Yaskawa INFORM job: OK_R2_O29-32(90,0_180)OKKR_HARDO.JBI

/JOB
//NAME OK_R2_O29-32(90,0_180)OKKR_HARDO
///FOLDERNAME X4
//POS
///NPOS 481,481,481,29,0,0
///TOOL 0
///POSTYPE PULSE
///PULSE
C00000=-97132,-107765,-123812,202,48316,-59447
C00001=-96375,-92560,-98278,-24892,54395,-33522
C00002=-118989,-99090,-96496,-10423,45001,-41425
C00003=-119482,-98696,-96132,-10013,44918,-41650
C00004=-120044,-95875,-95039,-9417,45618,-41989
C00005=-120040,-96488,-95280,-9446,45452,-41970
C00006=-120040,-96349,-93513,-9613,44449,-41863
C00007=-116902,-102455,-99217,-12157,45235,-40465
C00008=-92713,-84433,-91012,-29057,58273,-28062
C00009=-92713,-84514,-90161,-29225,57775,-27916
C00010=-92713,-84433,-91012,-29057,58273,-28062
C00011=-94031,-81016,-89513,-28080,58570,-28717
C00012=-92713,-84433,-91012,-29057,58273,-28062
C00013=-90703,-81163,-89579,-29929,59661,-27598
C00014=-92713,-84433,-91012,-29057,58273,-28062
C00015=-92432,-93178,-97379,-29384,57863,-27818
C00016=-124148,-115404,-96380,35354,30522,-76988
C00017=-124343,-116589,-99678,31918,27003,-75506
C00018=-121380,-108057,-94385,26950,26949,-73057
C00019=-119584,-104006,-91933,24006,26917,-71617
C00020=-119584,-103646,-90714,24467,26399,-71847
C00021=-119584,-104006,-91933,24006,26917,-71617
C00022=-119620,-100131,-90508,23194,27949,-71207
C00023=-120534,-102543,-91401,24964,27586,-72076
C00024=-122455,-107025,-93629,28318,27362,-73726
C00025=-122455,-106023,-90592,29616,26170,-74375
C00026=-120621,-104452,-90033,26656,25963,-72920
C00027=-122455,-106023,-90592,29616,26170,-74375
C00028=-124343,-116589,-99678,31918,27003,-75506
C00029=-121196,-113012,-111121,15968,43333,-61367
C00030=-113176,-99870,-108783,-18970,68338,-28733
C00031=-120594,-112521,-105960,-11204,51151,-28139
C00032=-122756,-104132,-102044,-9486,52748,-29227
C00033=-121295,-102030,-101271,-10379,53522,-28693
C00034=-122756,-104132,-102044,-9486,52748,-29227
C00035=-120055,-113496,-105331,-11710,50355,-27811
C00036=-117525,-106832,-103510,-13014,52989,-27048
C00037=-118169,-104316,-102602,-12476,53606,-27398
C00038=-117525,-106832,-103510,-13014,52989,-27048
C00039=-120055,-113496,-105331,-11710,50355,-27811
C00040=-122277,-105580,-101993,-9905,52039,-28956
C00041=-122277,-105483,-101030,-9979,51504,-28904
C00042=-122277,-105580,-101993,-9905,52039,-28956
C00043=-114234,-96976,-102629,-20681,62688,-27649
C00044=-111778,-96221,-107052,-21188,70616,-22267
C00045=-117350,-114999,-95956,-52919,38370,-55080
C00046=-108972,-69269,-80208,-51978,72625,-32902
C00047=-109543,-61925,-78651,-49562,78172,-29234
C00048=-109543,-62109,-77971,-49635,77832,-29052
C00049=-109543,-61925,-78651,-49562,78172,-29234
C00050=-110239,-61041,-78189,-49323,77924,-29446
C00051=-109543,-61925,-78651,-49562,78172,-29234
C00052=-107063,-66961,-84785,-50173,80254,-29118
C00053=-90901,-32599,-64406,-54667,92064,-27755
C00054=-92412,-28582,-59178,-54201,90556,-27610
C00055=-92412,-29145,-58034,-54170,89959,-27242
C00056=-92412,-28659,-59030,-54195,90478,-27561
C00057=-93599,-27197,-58027,-53876,89920,-27837
C00058=-92412,-28659,-59030,-54195,90478,-27561
C00059=-94015,-33926,-70364,-53928,92204,-29442
C00060=-96981,-29734,-65408,-52966,90116,-29668
C00061=-96981,-30385,-64512,-52944,89568,-29346
C00062=-96981,-29921,-65159,-52958,89962,-29578
C00063=-97341,-27509,-63519,-52853,89918,-29730
C00064=-96981,-29921,-65159,-52958,89962,-29578
C00065=-83985,-34763,-79826,-57770,100542,-29760
C00066=-119227,-121429,-124211,-4290,80037,5069
C00067=-103198,-96938,-112022,-8857,86341,9990
C00068=-104928,-94630,-110553,-8370,86444,9424
C00069=-105210,-91425,-109287,-8287,87275,9277
C00070=-105152,-92089,-109552,-8304,87105,9308
C00071=-105152,-92773,-108542,-8308,86142,9373
C00072=-104752,-96369,-111669,-8420,86257,9494
C00073=-93824,-83108,-104490,4346,83202,15848
C00074=-94227,-80625,-103370,4481,83809,15742
C00075=-95161,-74712,-100714,4798,85256,15503
C00076=-95037,-75505,-101078,4756,85066,15534
C00077=-95037,-76584,-99812,4762,83737,15482
C00078=-95852,-86288,-106522,5052,82929,15193
C00079=-119227,-121429,-124211,-4290,80037,5069
C00080=-108780,-117808,-111617,-31391,23506,27123
C00081=-87227,-129275,-103249,-15171,52693,43306
C00082=-62701,-112417,-81564,-27325,55133,54084
C00083=-102122,-48912,-69312,-5951,70900,35879
C00084=-115730,-7694,-35577,433,70873,-75154
C00085=-117065,58625,15220,1046,73703,-75581
C00086=-145520,63530,20841,13896,75272,-84857
C00087=-144593,33918,-9965,-2110,74261,-87786
C00088=-145469,31320,-10101,-1692,72990,-88049
C00089=-145469,30699,-8934,-1700,71953,-88037
C00090=-145469,30866,-9263,-1698,72241,-88041
C00091=-145880,26405,-13670,-1493,72653,-88180
C00092=-145880,26179,-13238,-1495,72270,-88176
C00093=-145579,28506,-10956,-1645,72067,-88074
C00094=-145661,28530,-12807,-1597,73217,-88116
C00095=-144591,77564,35073,-17956,86562,-90701
C00096=-144815,78144,37521,-17912,85364,-90602
C00097=-144815,77832,38454,-17925,84664,-90498
C00098=-144815,77924,38162,-17920,84880,-90530
C00099=-143930,80933,41834,-18166,84388,-90155
C00100=-143930,80814,42260,-18173,84080,-90109
C00101=-144274,79788,41005,-18076,84241,-90251
C00102=-144021,80584,40299,-18125,85099,-90292
C00103=-142778,71394,29201,-18425,87369,-90210
C00104=-142778,70963,30227,-18429,86558,-90088
C00105=-142778,71046,30015,-18428,86723,-90113
C00106=-141980,74470,34104,-18641,86176,-89759
C00107=-141980,74364,34402,-18643,85951,-89725
C00108=-142286,73285,33109,-18561,86114,-89854
C00109=-142258,74173,32193,-18559,87090,-89993
C00110=-151142,95382,53861,9912,94501,-89436
C00111=-151142,95214,54369,9904,94108,-89467
C00112=-151142,94960,55250,9895,93443,-89520
C00113=-151142,95064,54871,9900,93726,-89497
C00114=-151832,99566,60657,9969,92580,-89818
C00115=-151832,99473,61122,9966,92251,-89844
C00116=-151679,98392,59730,9950,92531,-89770
C00117=-151679,98651,58626,9962,93331,-89705
C00118=-139326,110012,65153,-7943,96581,-88072
C00119=-139426,116179,73372,-7897,94700,-87984
C00120=-139426,115886,74309,-7888,93978,-87938
C00121=-139426,116062,73720,-7895,94427,-87966
C00122=-140236,121957,81659,-7780,92511,-88115
C00123=-140236,121844,82405,-7775,91998,-88082
C00124=-140074,120418,80479,-7799,92463,-88057
C00125=-140074,120860,78539,-7816,93872,-88145
C00126=-141384,30046,-16215,-3642,76218,-86818
C00127=-144769,2915,-41310,-1997,77613,-87897
C00128=-120497,-21208,-21286,5945,66983,1716
C00129=-120331,-15331,-14033,5953,65534,1703
C00130=-120268,-12560,-10010,5981,64483,1671
C00131=-120268,-12013,-7946,6027,63500,1622
C00132=-120268,-12272,-8910,6006,63957,1643
C00133=-120268,-12272,-8910,6006,63957,1643
C00134=-120271,-10596,-7611,6006,64020,1643
C00135=-120265,-13710,-11092,5976,64558,1676
C00136=-121090,-15095,-12910,6234,65025,1394
C00137=-122392,-36893,-37139,6496,68816,1124
C00138=-103008,-20958,-23789,-34380,46191,-50944
C00139=-106920,-17705,-17148,-23301,36916,-65920
C00140=-100038,-3407,1736,-8309,24573,-69609
C00141=-100051,-3014,2749,-8424,24152,-69554
C00142=-100051,-2528,4297,-8659,23456,-69437
C00143=-99986,-3534,2326,-8528,24154,-69501
C00144=-100190,-1879,3683,-8197,24147,-69667
C00145=-100051,-3014,2749,-8424,24152,-69554
C00146=-107520,-15673,-12264,3373,26664,-75475
C00147=-107604,-14630,-9438,-26327,31803,-64502
C00148=-107301,-12783,-11511,-23446,35942,-65836
C00149=-106944,-14381,-11463,-24264,35264,-65385
C00150=-107257,-12837,-10189,-14623,32274,-69602
C00151=-111525,-14589,-10078,-816,28523,-72551
C00152=-98801,-12889,-18000,4905,35451,-65199
C00153=-115508,-28515,-28430,43638,36769,-74115
C00154=-104252,-46667,-49928,-23147,42547,-66097
C00155=-139326,111643,62701,-7999,98906,-88222
C00156=-140217,96503,46831,-7956,100791,-62986
C00157=-145074,69745,16622,-2645,91472,-63331
C00158=-144953,70943,20162,-2680,89915,-63261
C00159=-144922,69779,18776,-2690,90171,-63257
C00160=-144922,69779,18776,-2690,90171,-63257
C00161=-145083,66914,15382,-2644,90782,-63319
C00162=-137468,95477,49594,-19726,99949,-65005
C00163=-137749,101548,57639,-20808,101771,-65556
C00164=-141788,85517,37198,-20977,104871,-67541
C00165=-141788,85517,37198,-20977,104871,-67541
C00166=-141697,80573,32373,-24906,103800,-68015
C00167=-141133,64860,16683,-29804,96213,-66902
C00168=-143290,70938,23843,-29251,94388,-67208
C00169=-143290,72189,22259,-29351,95808,-67570
C00170=-136972,39162,-14968,-31401,103005,-67268
C00171=-136972,39162,-14968,-31401,103005,-67268
C00172=-104252,-46667,-49928,-23147,42547,-66097
C00173=-79661,-64382,-64322,-40022,51624,-56449
C00174=-25614,-129739,-89176,-60277,72547,-35569
C00175=-79661,-64382,-64322,-40022,51624,-56449
C00176=-120757,-91510,-125291,13460,57469,62186
C00177=-120699,-18778,-86977,11996,70937,63715
C00178=-120626,-71428,-80514,17274,40782,59546
C00179=-119608,-71223,-77796,25261,41295,55541
C00180=-118939,-66183,-73787,24596,41210,55877
C00181=-120629,-71631,-77769,17920,39069,59168
C00182=-120359,-74344,-77822,18174,37713,59000
C00183=-130492,-64065,-72622,39267,48666,48449
C00184=-128767,-64530,-72039,39655,46741,50471
C00185=-122213,-56683,-67868,39757,48514,50554
C00186=-119025,-61972,-83652,25821,56823,82211
C00187=-119200,-79046,-90724,17013,50162,51422
C00188=-120627,-71422,-82568,-22551,39281,-72893
C00189=-120626,-71781,-79821,-23470,37548,-72366
C00190=-120451,-70478,-78279,-23795,37340,-72196
C00191=-120359,-74605,-80000,-24468,36394,-71829
C00192=-120633,-71786,-79901,-23439,37590,-72383
C00193=-120966,-71169,-78914,-23220,37205,-72458
C00194=-120627,-71746,-82478,-22655,39075,-72833
C00195=-120628,-68509,-91693,-24468,73270,-29259
C00196=-120628,-69110,-90711,-24576,72437,-29080
C00197=-120650,-67557,-87939,-24676,71616,-28918
C00198=-120635,-69084,-90779,-24566,72485,-29092
C00199=-120360,-72648,-91234,-24892,71146,-28701
C00200=-102891,-55002,-81397,-31881,79379,-24336
C00201=-98614,-51013,-79162,-33441,81477,-23356
C00202=-110216,-66091,-87232,-17856,68486,-33346
C00203=-120628,-67132,-93536,-6272,76376,-26037
C00204=-120629,-65307,-95540,-6224,78533,-26146
C00205=-125976,-49581,-89047,24033,107700,-27220
C00206=-114932,-69047,-98963,12803,96211,-16970
C00207=-121913,-67019,-96424,19539,98441,-21657
C00208=-120636,-64508,-96476,19357,99419,-21079
C00209=-115636,-66806,-97970,12989,96839,-17125
C00210=-122763,-41192,-84008,14889,102356,-18715
C00211=-119690,-45533,-86635,11059,99611,-14244
C00212=-123247,-59553,-98781,12453,98224,-12183
C00213=-120629,-65231,-95763,5470,82909,-26902
C00214=-114225,-78059,-113057,2895,86652,-24852
C00215=-100902,-64627,-95050,-11985,78171,-15678
C00216=-98861,-75542,-94548,-15732,66869,-13224
C00217=-119874,-71154,-93232,19306,73218,3187
C00218=-121912,-70007,-92672,20214,73908,2597
C00219=-98680,-77069,-90223,-16254,63590,-12696
C00220=-96345,-50788,-86680,-18048,88539,-14542
C00221=-93223,-76561,-100164,-23339,71866,-11449
C00222=-120630,-61713,-98239,-7195,94993,11495
C00223=-120629,-64150,-96408,-7165,92633,11631
C00224=-127375,-45154,-88676,-4909,106126,9193
C00225=-120636,-64104,-96466,-7164,92690,11625
C00226=-119876,-67808,-97008,-7371,91195,11945
C00227=-122268,-40179,-85765,-5907,107177,10698
C00228=-117984,-41448,-85856,-6781,104340,12121
C00229=-117785,-40415,-85699,-6838,104785,12155
C00230=-118921,-47757,-88901,-6950,100752,11907
C00231=-128083,-66216,-96645,-288,90786,4689
C00232=-127344,-66265,-96731,-512,90816,4915
C00233=-120629,-63706,-96407,-7167,92858,11618
C00234=-119771,-61779,-98541,-7450,95212,11740
C00235=-113204,-65987,-111954,-20711,103856,-62714
C00236=-120630,-56479,-101004,-18441,100644,-64439
C00237=-137856,-73372,-107086,809,89532,-64747
C00238=-119374,-56629,-99297,-18722,99813,-63925
C00239=-120637,-56952,-100808,-18413,100297,-64387
C00240=-141222,-46996,-93568,2005,94815,-65665
C00241=-144586,-98422,-105395,6853,55489,-67509
C00242=-126129,-101623,-112002,-18280,57665,-60270
C00243=-107171,-88917,-111068,-40561,70673,-56675
C00244=-99343,-43314,-99502,-42439,86261,-59904
C00245=-52791,5163,-64646,-46831,92051,-59410
C00246=3643,-76224,-106676,19950,71810,76872
C00247=-31759,-97415,-96886,-14116,45711,48381
C00248=-44548,-99394,-97233,-12419,44266,52870
C00249=-91182,-106612,-98498,-6229,38996,69241
C00250=-120252,-111112,-99286,-2370,35711,79446
C00251=-120252,-111112,-99286,-2370,35711,79446
C00252=-122061,-111349,-89048,-12693,25666,-59648
C00253=-121671,-62095,-66353,-9610,36862,-61269
C00254=-121347,-21258,-21397,-11816,30334,-60091
C00255=-120891,-15529,-14207,-12963,28955,-59505
C00256=-120717,-13203,-11253,-13455,28377,-59255
C00257=-120568,-11431,-9889,-13625,28472,-59171
C00258=-120717,-13203,-11253,-13455,28377,-59255
C00259=-120696,-12930,-10087,-13737,27819,-59112
C00260=-120692,-12567,-8711,-14046,27176,-58956
C00261=-120696,-12930,-10087,-13737,27819,-59112
C00262=-120870,-15275,-13061,-13229,28399,-59370
C00263=-123043,5425,8644,-60342,36239,-52197
C00264=-124447,11447,16156,-60569,34992,-52124
C00265=-124447,11983,17788,-61490,34623,-51621
C00266=-127145,7414,15485,-62450,27197,-51222
C00267=-127103,8624,16548,-62533,27208,-51178
C00268=-127127,7743,15901,-62612,27166,-51140
C00269=-124895,-3553,-1899,-45295,28876,-55547
C00270=-121324,-21046,-20294,-12047,29779,-59971
C00271=-121671,-62095,-66353,-9610,36862,-61269
C00272=-122061,-111349,-89048,-12693,25666,-59648
C00273=-120249,-110580,-95500,-2498,33656,79516
C00274=-120367,-55464,-65807,-1899,43695,79179
C00275=-120372,-19909,-20534,-2331,34109,79427
C00276=-120603,-14858,-13386,-2171,32301,79344
C00277=-118432,-12836,-10242,-4853,31501,80756
C00278=-118432,-12391,-8558,-4969,30699,80814
C00279=-118432,-12586,-9286,-4918,31044,80789
C00280=-118432,-12586,-9286,-4918,31044,80789
C00281=-118451,-11211,-8225,-4888,31096,80773
C00282=-120719,-12556,-10288,-2076,31575,79294
C00283=-120630,-14625,-13229,-2138,32324,79327
C00284=-131566,-7566,-2012,56880,47864,36778
C00285=-127270,2858,10417,64219,55978,24180
C00286=-127270,2872,10457,64230,55970,24171
C00287=-127270,3275,11649,64548,55732,23910
C00288=-127279,2816,10434,64241,55969,24162
C00289=-127226,4202,11617,64241,55929,24162
C00290=-127288,2760,10411,64252,55968,24153
C00291=-139196,1750,6280,64814,64625,23032
C00292=-119950,-29718,-27457,-2865,33344,79709
C00293=-120367,-55464,-65807,-1899,43695,79179
C00294=-120071,-144849,-99630,-4685,18622,80601
C00295=-120101,-156003,-112174,-4198,20603,80368
C00296=-118703,-129435,-118376,-15737,33464,74082
C00297=-118229,-124990,-122609,-18843,37087,72450
C00298=-117709,-116078,-100914,-29615,27785,74634
C00299=-121884,-95901,-99968,19866,48605,45126
C00300=-120671,-70136,-84949,27990,60023,38564
C00301=-120478,-67274,-83298,27761,60367,38737
C00302=-120671,-68730,-84259,27912,60289,38637
C00303=-120481,-64965,-83246,27119,62754,39366
C00304=-120481,-65408,-81931,27360,61828,39126
C00305=-121686,-66768,-84557,27809,63026,38954
C00306=-141024,-58078,-80968,36822,71957,33892
C00307=-140832,-52974,-76512,36762,71783,33908
C00308=-140832,-53417,-75497,36922,71094,33665
C00309=-140832,-52974,-76512,36762,71783,33908
C00310=-140279,-50808,-75283,36453,71852,34159
C00311=-140832,-52974,-76512,36762,71783,33908
C00312=-109942,-69794,-83321,-14013,53448,56252
C00313=-112063,-69620,-83237,-12481,53147,55418
C00314=-109971,-72059,-85461,-13968,53588,56219
C00315=-110807,-74146,-92563,-12442,56365,55924
C00316=-138671,-88440,-95611,17208,48170,52520
C00317=-138671,-88615,-94297,17448,47310,52358
C00318=-138671,-88440,-95611,17208,48170,52520
C00319=-138502,-86929,-95389,16910,48750,52704
C00320=-138041,-84511,-94358,16397,49242,52997
C00321=-138502,-86929,-95389,16910,48750,52704
C00322=-119374,-94871,-99184,-14699,45596,69062
C00323=-119374,-95024,-95430,-15324,43285,69457
C00324=-120961,-93958,-95008,-13845,43283,68674
C00325=-119374,-95024,-95430,-15324,43285,69457
C00326=-119544,-103546,-104622,-14834,44490,69166
C00327=-118175,-83390,-115370,-9254,78664,2265
C00328=-136131,-54129,-95643,4560,92395,119
C00329=-136131,-54129,-95643,4560,92395,119
C00330=-136131,-54129,-95643,4560,92395,119
C00331=-136131,-55910,-94548,4553,90811,61
C00332=-136131,-54129,-95643,4560,92395,119
C00333=-118826,-50989,-93921,-11407,94620,13199
C00334=-119876,-53326,-92440,-11017,92423,13086
C00335=-120690,-52300,-91874,-10745,92506,12834
C00336=-119876,-53326,-92440,-11017,92423,13086
C00337=-118826,-50270,-94307,-11422,95216,13144
C00338=-141793,-55820,-97332,7512,93105,-2300
C00339=-140356,-59957,-95696,6990,89886,-2061
C00340=-139743,-58912,-95151,6779,90039,-1868
C00341=-140356,-59957,-95696,6990,89886,-2061
C00342=-140356,-55082,-98612,7026,94155,-1823
C00343=-131844,-82412,-106901,19181,77049,14413
C00344=-121763,-121440,-108343,34263,48676,32319
C00345=-121436,-111193,-102207,33362,49794,32929
C00346=-120328,-103716,-97102,32376,49958,33559
C00347=-120328,-103424,-95545,32743,49272,33305
C00348=-120328,-103597,-96437,32532,49662,33450
C00349=-119706,-101713,-95741,31911,49887,33849
C00350=-120328,-103597,-96437,32532,49662,33450
C00351=-120421,-109652,-101209,32668,49551,33360
C00352=-120678,-119715,-107328,33483,48463,32809
C00353=-145717,-65257,-81010,41655,68644,28827
C00354=-145541,-64355,-79967,41625,68428,28817
C00355=-145541,-64661,-78699,41864,67717,28513
C00356=-145541,-64450,-79596,41693,68217,28727
C00357=-144419,-63348,-79027,41165,67869,29094
C00358=-145541,-64450,-79596,41693,68217,28727
C00359=-144489,-68274,-88356,40433,70363,30088
C00360=-140701,-65348,-85833,38739,68695,31071
C00361=-140701,-65803,-84785,38949,68003,30804
C00362=-140701,-65400,-85721,38761,68620,31042
C00363=-140042,-62987,-84490,38345,68721,31364
C00364=-140701,-65400,-85721,38761,68620,31042
C00365=-129105,-89797,-100104,-8257,42122,-63791
C00366=-127638,-62786,-75319,-9961,40926,-62941
C00367=-127541,-60842,-73212,-10119,40642,-62858
C00368=-127452,-58887,-72168,-10136,41010,-62858
C00369=-127541,-60842,-73212,-10119,40642,-62858
C00370=-127484,-59721,-71596,-10263,40237,-62779
C00371=-127484,-59825,-70645,-10399,39608,-62699
C00372=-127484,-59721,-71596,-10263,40237,-62779
C00373=-128516,-69367,-82634,-8882,41931,-63486
C00374=-136804,-49406,-65089,-22327,37576,-67328
C00375=-138093,-44400,-58341,-21720,35770,-67534
C00376=-137893,-42671,-57282,-21821,36047,-67500
C00377=-138034,-43342,-57719,-21701,35939,-67550
C00378=-137984,-43593,-56312,-22278,35025,-67233
C00379=-137984,-43463,-57769,-21774,35919,-67515
C00380=-121497,-78215,-85327,-19946,40083,-59616
C00381=-120626,-71657,-80701,-17243,40860,-59361
C00382=-126255,-72821,-79643,-11943,38658,-61920
C00383=-124460,-69554,-75696,-14032,38208,-60874
C00384=-120888,-74575,-78008,-18145,37790,-58814
C00385=-120633,-71857,-77956,-17876,39147,-58988
C00386=-120627,-71204,-76479,-18098,38609,-58863
C00387=-136164,-60832,-69738,-17624,37003,-72099
C00388=-124488,-74552,-79755,-29777,39497,-66170
C00389=-118213,-106277,-106559,-35084,42029,-63565
C00390=-120627,-70570,-83191,7863,37643,76584
C00391=-120626,-71021,-80486,8216,35764,76386
C00392=-117835,-70487,-78994,2708,35489,78081
C00393=-120887,-73898,-80698,8807,34458,76086
C00394=-120633,-71014,-80560,8214,35814,76388
C00395=-120357,-69871,-78574,5676,35674,76676
C00396=-149434,-47635,-66681,32878,46415,64025
C00397=-156080,-38551,-61157,37208,50074,62118
C00398=-120626,-71358,-80242,8280,35444,76351
C00399=-120627,-70947,-82965,7922,37313,76550
C00400=-120635,-68263,-89533,19357,55237,54189
C00401=-120627,-69277,-87249,27960,61590,38909
C00402=-120627,-70131,-84728,28472,59826,38424
C00403=-119745,-63249,-82789,26446,65626,40301
C00404=-120887,-73269,-85067,29013,58674,37985
C00405=-120633,-70114,-84797,28462,59873,38435
C00406=-120443,-58955,-81680,26193,68992,40844
C00407=-137016,-48093,-75675,33483,76149,36536
C00408=-111378,-73522,-86374,8880,55488,45224
C00409=-108292,-90151,-101040,6716,55677,46453
C00410=-104551,-107393,-114036,4170,54574,47870
C00411=-131132,-52506,-88181,-2999,76585,58563
C00412=-128416,-45796,-82269,-5250,83117,42213
C00413=-120634,-69367,-86746,-19850,61513,61572
C00414=-119352,-71200,-86390,-20819,60725,62219
C00415=-124049,-46051,-81029,-10377,81461,42067
C00416=-121481,-32611,-71357,-8547,80518,38471
C00417=-129432,-34048,-72513,3927,79787,30181
C00418=-133185,-27484,-76607,10911,90885,32661
C00419=-131562,-31841,-87200,10336,94922,33460
C00420=-120628,-67882,-90305,8002,60955,27137
C00421=-120628,-68780,-88641,8118,59484,27029
C00422=-119184,-68852,-87338,7230,58521,27500
C00423=-119351,-70586,-88688,7347,58476,27433
C00424=-121372,-71710,-89222,8706,58421,26669
C00425=-119224,-70326,-83140,7530,55210,27256
C00426=-118796,-48871,-84615,7155,80182,30422
C00427=-125592,-51833,-97720,10091,87276,28906
C00428=-113783,-56439,-81210,15698,57996,69309
C00429=-107790,-54952,-79381,11557,56703,71425
C00430=-114138,-25426,-67877,22136,88341,34287
C00431=-121370,-73680,-74765,39382,39185,61177
C00432=-120632,-71435,-74935,37828,39854,62032
C00433=-120118,-28476,-67262,26234,84322,31994
C00434=-128183,-20881,-60116,35034,87592,29156
C00435=-128620,-20492,-59969,35459,87655,29119
C00436=-131561,-17349,-57221,36148,87598,28432
C00437=-145073,1746,-39674,39691,86205,25187
C00438=-146718,4880,-36652,40179,85809,24767
C00439=-152046,17466,-29664,47680,97969,20185
C00440=-155175,14277,-38805,49221,102130,20939
C00441=-135677,-24502,-83351,29476,105612,50888
C00442=-120631,-49325,-102634,14154,102303,71085
C00443=-120630,-54638,-100904,13945,98616,70657
C00444=-113110,-76964,-106909,6133,84021,70452
C00445=-120637,-55119,-100712,13931,98263,70614
C00446=-121882,-54885,-99226,14292,97671,70180
C00447=-108261,-50195,-93515,4199,89241,72102
C00448=-118173,-67191,-91447,22538,66327,68916
C00449=-120627,-69075,-88308,30031,58405,66774
C00450=-120628,-67609,-91029,29341,60528,67400
C00451=-120651,-137986,-128118,34242,49089,63541
C00452=-120704,-83666,-109294,28636,63184,68115
C00453=-120704,-83666,-109294,28636,63184,68115
C00454=-122061,-111349,-89048,-12693,25666,-59648
C00455=-121671,-62095,-66353,-9610,36862,-61269
C00456=-120675,-12683,-10165,-1101,31339,-85533
C00457=-117312,-15222,-7734,-15098,24829,-82061
C00458=-120855,-14769,-11753,-884,31242,-85646
C00459=-120680,-13066,-11724,-1072,32101,-85548
C00460=-110921,-9380,-5536,-39323,36544,-54600
C00461=-105611,16644,27067,-74678,55970,-29641
C00462=-105060,15092,17806,-65581,60394,-35506
C00463=-113952,17541,-9445,-35713,50265,-81352
C00464=-121726,-68659,-62259,-14447,23269,-58731
C00465=-122061,-111349,-89048,-12693,25666,-59648
C00466=-120249,-110580,-95500,-2498,33656,79516
C00467=-120367,-55464,-65807,-1899,43695,79179
C00468=-123079,18123,-5334,37346,69821,35077
C00469=-120790,5622,-11235,35661,58510,35599
C00470=-123082,18120,-5282,37355,69796,35066
C00471=-123254,15918,-6072,37557,69350,34829
C00472=-101635,-726,-13913,25769,46964,40903
C00473=-122250,26655,19444,63036,59530,30813
C00474=-129965,36435,30593,70202,68747,28349
C00475=-135677,36825,21549,57633,74723,28944
C00476=-134949,-3767,-37487,36447,81076,35091
C00477=-139267,-30752,-53917,52477,61088,25483
C00478=-156581,-111669,-93710,65875,62680,14502
C00479=-153491,-118067,-95704,59271,58057,20364
C00480=-32064,-128753,-95704,15399,77815,-718
BC00000=40633,757095,1075175
BC00001=40600,786248,1075175
BC00002=40600,786248,1075175
BC00003=40600,786248,1075175
BC00004=40600,786248,1075175
BC00005=40600,786248,1075175
BC00006=40600,786248,1075175
BC00007=40600,786248,1075175
BC00008=40594,791778,1075175
BC00009=40594,791778,1075175
BC00010=40594,791778,1075175
BC00011=40594,791778,1075175
BC00012=40594,791778,1075175
BC00013=40594,791778,1075175
BC00014=40594,791778,1075175
BC00015=40594,791778,1075175
BC00016=40594,791778,1075175
BC00017=50995,786704,1075175
BC00018=50995,786704,1075175
BC00019=50995,786704,1075175
BC00020=50995,786704,1075175
BC00021=50995,786704,1075175
BC00022=50995,786704,1075175
BC00023=50995,786704,1075175
BC00024=50995,786704,1075175
BC00025=50995,786704,1075175
BC00026=50995,786704,1075175
BC00027=50995,786704,1075175
BC00028=50995,786704,1075175
BC00029=64165,785759,1075175
BC00030=97726,783351,1075175
BC00031=97726,783351,1075175
BC00032=97726,783351,1075175
BC00033=97726,783351,1075175
BC00034=97726,783351,1075175
BC00035=97726,783351,1075175
BC00036=97726,783351,1075175
BC00037=97726,783351,1075175
BC00038=97726,783351,1075175
BC00039=97726,783351,1075175
BC00040=97726,783351,1075175
BC00041=97726,783351,1075175
BC00042=97726,783351,1075175
BC00043=97726,783351,1075175
BC00044=97726,783351,1075175
BC00045=161258,787851,1075175
BC00046=161258,787851,1075175
BC00047=161258,787851,1075175
BC00048=161258,787851,1075175
BC00049=161258,787851,1075175
BC00050=161258,787851,1075175
BC00051=161258,787851,1075175
BC00052=161258,787851,1075175
BC00053=161258,787851,1075175
BC00054=161258,787851,1075175
BC00055=161258,787851,1075175
BC00056=161258,787851,1075175
BC00057=161258,787851,1075175
BC00058=161258,787851,1075175
BC00059=161258,787851,1075175
BC00060=161258,787851,1075175
BC00061=161258,787851,1075175
BC00062=161258,787851,1075175
BC00063=161258,787851,1075175
BC00064=161258,787851,1075175
BC00065=161258,787851,1075175
BC00066=272656,866721,1075175
BC00067=272656,866721,1075175
BC00068=272656,866721,1075175
BC00069=272656,866721,1075175
BC00070=272656,866721,1075175
BC00071=272656,866721,1075175
BC00072=272656,866721,1075175
BC00073=272656,866721,1075175
BC00074=272656,866721,1075175
BC00075=272656,866721,1075175
BC00076=272656,866721,1075175
BC00077=272656,866721,1075175
BC00078=272656,866721,1075175
BC00079=272656,866721,1075175
BC00080=276508,696729,1075050
BC00081=283938,685942,1074810
BC00082=283938,717840,610142
BC00083=283938,747609,176485
BC00084=283938,747609,176485
BC00085=283938,747609,53405
BC00086=343059,747609,53405
BC00087=343059,747609,53405
BC00088=343059,747609,53405
BC00089=343059,747609,53405
BC00090=343059,747609,53405
BC00091=343059,747609,53405
BC00092=343059,747609,53405
BC00093=343059,747609,53405
BC00094=343059,747609,53405
BC00095=343059,747609,53405
BC00096=343059,747609,53405
BC00097=343059,747609,53405
BC00098=343059,747609,53405
BC00099=343059,747609,53405
BC00100=343059,747609,53405
BC00101=343059,747609,53405
BC00102=343059,747609,53405
BC00103=343059,747609,53405
BC00104=343059,747609,53405
BC00105=343059,747609,53405
BC00106=343059,747609,53405
BC00107=343059,747609,53405
BC00108=343059,747609,53405
BC00109=343059,747609,53405
BC00110=343059,747609,53405
BC00111=343059,747609,53405
BC00112=343059,747609,53405
BC00113=343059,747609,53405
BC00114=343059,747609,53405
BC00115=343059,747609,53405
BC00116=343059,747609,53405
BC00117=343059,747609,53405
BC00118=343059,747609,24
BC00119=343059,747609,24
BC00120=343059,747609,24
BC00121=343059,747609,24
BC00122=343059,747609,24
BC00123=343059,747609,24
BC00124=343059,747609,24
BC00125=343059,747609,24
BC00126=343059,747609,53405
BC00127=343059,747609,53405
BC00128=272784,788172,221315
BC00129=272784,788172,221315
BC00130=272784,788172,221315
BC00131=272784,788172,221315
BC00132=272784,788172,221315
BC00133=272784,788172,221315
BC00134=272784,788172,221315
BC00135=272784,788172,221315
BC00136=272784,788172,221315
BC00137=272784,788172,221315
BC00138=262280,759997,129875
BC00139=260494,755206,114324
BC00140=260786,755989,116866
BC00141=260786,755989,116866
BC00142=260786,755989,116866
BC00143=260786,755989,116866
BC00144=260786,755989,116866
BC00145=260786,755989,116866
BC00146=260786,755989,116866
BC00147=260462,756705,106964
BC00148=260456,756989,105568
BC00149=260456,756989,105568
BC00150=253777,756505,101682
BC00151=288441,762581,102049
BC00152=263875,774786,46208
BC00153=263467,774501,47249
BC00154=260494,755206,114324
BC00155=343059,747609,24
BC00156=344552,769122,24
BC00157=344552,769122,24
BC00158=344552,769122,24
BC00159=344552,769122,24
BC00160=344552,769122,24
BC00161=344552,769122,24
BC00162=344552,769122,24
BC00163=344552,769122,24
BC00164=344552,769122,24
BC00165=344552,769122,24
BC00166=344552,769122,24
BC00167=344552,769122,24
BC00168=344552,769122,24
BC00169=344552,769122,24
BC00170=344552,769122,24
BC00171=344552,769122,24
BC00172=260494,755206,114324
BC00173=260494,678873,114324
BC00174=260494,678873,389237
BC00175=260494,678873,1074810
BC00176=249358,694721,1075175
BC00177=249358,736986,1075175
BC00178=249358,791546,1075175
BC00179=248933,799175,1075175
BC00180=248933,799175,1075175
BC00181=248933,799175,1075175
BC00182=248933,799175,1075175
BC00183=303936,808747,1075173
BC00184=301664,808908,1075173
BC00185=301664,808908,1075173
BC00186=278558,810544,1075175
BC00187=259247,802769,1075175
BC00188=179692,770739,1075175
BC00189=178037,775961,1075175
BC00190=177375,778050,1075175
BC00191=177375,778050,1075175
BC00192=177375,778050,1075175
BC00193=105009,765455,1075171
BC00194=106185,757956,1075175
BC00195=70430,778998,1075175
BC00196=70141,784459,1075175
BC00197=70031,786589,1075172
BC00198=70026,786643,1075175
BC00199=70026,786643,1075175
BC00200=71134,786838,1075175
BC00201=71134,786838,1075175
BC00202=71134,786838,1075175
BC00203=80371,790898,1075175
BC00204=79285,785365,1075175
BC00205=47064,807646,1075175
BC00206=47064,807646,1075175
BC00207=47306,807824,1075175
BC00208=47306,807824,1075175
BC00209=47064,807646,1075175
BC00210=47064,807646,1075175
BC00211=47064,807646,1075175
BC00212=47064,807646,1075175
BC00213=54175,793583,1075175
BC00214=54175,793583,1075175
BC00215=54992,769398,1075175
BC00216=54992,769398,1075175
BC00217=54992,769398,1075175
BC00218=54992,769398,1075175
BC00219=54992,769398,1075175
BC00220=54992,769398,1075175
BC00221=54992,769398,1075175
BC00222=110304,782517,1075175
BC00223=108105,787545,1075175
BC00224=107226,789556,1075175
BC00225=107226,789556,1075175
BC00226=107226,789556,1075175
BC00227=107226,789556,1075175
BC00228=107227,789556,1075174
BC00229=107227,789556,1075174
BC00230=127545,800970,1075174
BC00231=170992,825380,1075175
BC00232=170992,825380,1075175
BC00233=172064,823477,1075175
BC00234=174263,818448,1075175
BC00235=118984,806720,1075175
BC00236=118671,807322,1075175
BC00237=118546,807563,1075175
BC00238=118546,807563,1075175
BC00239=118546,807563,1075175
BC00240=118546,807563,1075175
BC00241=118546,807563,1075175
BC00242=125414,796325,1075175
BC00243=133048,783833,1075175
BC00244=133048,783833,1075175
BC00245=133048,671052,1075175
BC00246=199464,674570,1075173
BC00247=264750,673287,320956
BC00248=270450,673384,288313
BC00249=291235,673736,169281
BC00250=304191,673956,95082
BC00251=304191,673956,95082
BC00252=164726,705512,84367
BC00253=164726,728796,84367
BC00254=164726,745774,84367
BC00255=164726,745774,84367
BC00256=164726,745774,84367
BC00257=164726,745774,84367
BC00258=164726,745774,84367
BC00259=164726,745774,84367
BC00260=164726,745774,84367
BC00261=164726,745774,84367
BC00262=164726,745774,84367
BC00263=164726,745774,84367
BC00264=164726,745774,84367
BC00265=164726,745774,84367
BC00266=164726,745774,84367
BC00267=164726,745774,84367
BC00268=164726,745774,84367
BC00269=164726,745774,84367
BC00270=164726,745774,84367
BC00271=164726,728796,84367
BC00272=164726,705512,84367
BC00273=304191,706504,95082
BC00274=304191,706504,95082
BC00275=304191,726145,95082
BC00276=304191,726145,95082
BC00277=304191,726145,95082
BC00278=304191,726145,95082
BC00279=304191,726145,95082
BC00280=304191,726145,95082
BC00281=304191,726145,95082
BC00282=304191,726145,95082
BC00283=304191,726145,95082
BC00284=304191,726145,95082
BC00285=304191,726145,95082
BC00286=304191,726145,95082
BC00287=304191,726145,95082
BC00288=304191,726145,95082
BC00289=304191,726145,95082
BC00290=304191,726145,95082
BC00291=304191,726145,95082
BC00292=304191,726145,95082
BC00293=304191,706504,95082
BC00294=304191,706504,95082
BC00295=304191,706504,1074810
BC00296=355942,722834,1075048
BC00297=369200,753216,1075109
BC00298=383735,786522,1075175
BC00299=370224,778181,1075175
BC00300=364232,774482,1075175
BC00301=364232,774482,1075175
BC00302=364232,774482,1075175
BC00303=364232,774482,1075175
BC00304=364232,774482,1075175
BC00305=364232,774482,1075175
BC00306=364232,774482,1075175
BC00307=364232,774482,1075175
BC00308=364232,774482,1075175
BC00309=364232,774482,1075175
BC00310=364232,774482,1075175
BC00311=364232,774482,1075175
BC00312=364232,774482,1075175
BC00313=364232,774482,1075175
BC00314=364232,774482,1075175
BC00315=365231,775099,1075175
BC00316=383734,786522,1075172
BC00317=383734,786522,1075172
BC00318=383734,786522,1075172
BC00319=383734,786522,1075172
BC00320=383734,786522,1075172
BC00321=383734,786522,1075172
BC00322=383735,786522,1075175
BC00323=383735,786522,1075175
BC00324=383735,786522,1075175
BC00325=383735,786522,1075175
BC00326=383735,786522,1075175
BC00327=375764,783819,1075175
BC00328=375764,783819,1075175
BC00329=375764,783819,1075175
BC00330=375764,783819,1075175
BC00331=375764,783819,1075175
BC00332=375764,783819,1075175
BC00333=375764,783819,1075175
BC00334=375764,783819,1075175
BC00335=375764,783819,1075175
BC00336=375764,783819,1075175
BC00337=375764,783819,1075175
BC00338=375764,783819,1075175
BC00339=375764,783819,1075175
BC00340=375764,783819,1075175
BC00341=375764,783819,1075175
BC00342=375764,783819,1075175
BC00343=337318,787163,1075175
BC00344=291781,791124,1075175
BC00345=291781,791124,1075175
BC00346=291781,791124,1075175
BC00347=291781,791124,1075175
BC00348=291781,791124,1075175
BC00349=291781,791124,1075175
BC00350=291781,791124,1075175
BC00351=291781,791124,1075175
BC00352=291781,791124,1075175
BC00353=291781,791124,1075175
BC00354=291781,791124,1075175
BC00355=291781,791124,1075175
BC00356=291781,791124,1075175
BC00357=291781,791124,1075175
BC00358=291781,791124,1075175
BC00359=291781,791124,1075175
BC00360=291781,791124,1075175
BC00361=291781,791124,1075175
BC00362=291781,791124,1075175
BC00363=291781,791124,1075175
BC00364=291781,791124,1075175
BC00365=187451,791796,1075175
BC00366=187451,791796,1075175
BC00367=187451,791796,1075175
BC00368=187451,791796,1075175
BC00369=187451,791796,1075175
BC00370=187451,791796,1075175
BC00371=187451,791796,1075175
BC00372=187451,791796,1075175
BC00373=187451,791796,1075175
BC00374=187451,791796,1075175
BC00375=187451,791796,1075175
BC00376=187451,791796,1075175
BC00377=187451,791796,1075175
BC00378=187451,791796,1075175
BC00379=187451,791796,1075175
BC00380=187451,791796,1075175
BC00381=187451,791796,1075175
BC00382=187781,797245,1075175
BC00383=187913,799425,1075175
BC00384=187913,799425,1075175
BC00385=187913,799425,1075175
BC00386=132893,808904,1075175
BC00387=158479,810741,1075175
BC00388=158479,810741,1075175
BC00389=158479,810741,1075175
BC00390=350755,754943,1075175
BC00391=351085,760393,1075175
BC00392=351217,762573,1075175
BC00393=351217,762573,1075175
BC00394=351217,762573,1075175
BC00395=351217,762573,1075175
BC00396=351217,762573,1075175
BC00397=351217,762573,1075175
BC00398=274278,773616,1075175
BC00399=273948,768166,1075175
BC00400=328759,768723,1075175
BC00401=363745,769079,1075175
BC00402=364075,774529,1075175
BC00403=364207,776708,1075175
BC00404=364207,776708,1075175
BC00405=364207,776708,1075175
BC00406=359505,777527,1075175
BC00407=359505,777527,1075175
BC00408=331768,783965,1075175
BC00409=331768,783965,1075175
BC00410=331768,783965,1075175
BC00411=392812,762505,1075175
BC00412=387447,767589,1075164
BC00413=386542,767124,1075175
BC00414=386542,767124,1075175
BC00415=387446,767590,1075167
BC00416=387446,767590,1075168
BC00417=387446,767590,1075168
BC00418=387446,767590,1075168
BC00419=387446,767590,1075168
BC00420=342059,744861,1075175
BC00421=340306,751293,1075175
BC00422=339605,753866,1075175
BC00423=339605,753866,1075175
BC00424=339605,753866,1075175
BC00425=339643,753874,1075175
BC00426=339648,753875,1075175
BC00427=339648,753875,1075175
BC00428=300304,742240,1075175
BC00429=300304,742240,1075175
BC00430=303441,749269,1075175
BC00431=303441,749269,1075175
BC00432=303441,749269,1075175
BC00433=303441,749269,1075175
BC00434=303441,749269,1075175
BC00435=303441,749269,1075175
BC00436=303441,749269,1075175
BC00437=303441,749269,1075175
BC00438=303441,749269,1075175
BC00439=303441,749269,1075175
BC00440=303441,749269,1075175
BC00441=315359,779867,1075175
BC00442=323854,801676,1075175
BC00443=324239,802262,1075175
BC00444=324392,802497,1075175
BC00445=324392,802497,1075175
BC00446=324392,802497,1075175
BC00447=324392,802497,1075175
BC00448=317597,791028,1075175
BC00449=312615,782697,1075175
BC00450=310293,778880,1075175
BC00451=310293,778880,1075175
BC00452=310293,671436,1075175
BC00453=310293,671436,96460
BC00454=164726,705512,84367
BC00455=164726,728796,84367
BC00456=159129,750828,110218
BC00457=158936,752443,102455
BC00458=158913,752632,101547
BC00459=158913,752632,101547
BC00460=118735,759517,101182
BC00461=118735,759517,101182
BC00462=118735,759517,101182
BC00463=151265,712492,23474
BC00464=164726,728796,84367
BC00465=164726,705512,84367
BC00466=304191,706504,95082
BC00467=304191,706504,95082
BC00468=252242,721798,53
BC00469=252847,723541,52
BC00470=252870,723608,53
BC00471=252870,723608,53
BC00472=252847,723541,52
BC00473=303936,700545,53
BC00474=303936,700545,53
BC00475=303936,700545,53
BC00476=292348,710053,53
BC00477=292348,710053,53
BC00478=292348,710053,53
BC00479=293342,710891,8032
BC00480=241772,668348,8032
EC00000=-798156,1112951
EC00001=-798156,1112951
EC00002=-798156,1112951
EC00003=-798156,1112951
EC00004=-798156,1112951
EC00005=-798156,1112951
EC00006=-798156,1112951
EC00007=-798156,1112951
EC00008=-798156,1112951
EC00009=-798156,1112951
EC00010=-798156,1112951
EC00011=-798156,1112951
EC00012=-798156,1112951
EC00013=-798156,1112951
EC00014=-798156,1112951
EC00015=-798156,1112951
EC00016=-798156,1112951
EC00017=-798156,1112951
EC00018=-798156,1112951
EC00019=-798156,1112951
EC00020=-798156,1112951
EC00021=-798156,1112951
EC00022=-798156,1112951
EC00023=-798156,1112951
EC00024=-798156,1112951
EC00025=-798156,1112951
EC00026=-798156,1112951
EC00027=-798156,1112951
EC00028=-798156,1112951
EC00029=-798156,1112951
EC00030=-798156,1112951
EC00031=-798156,1112951
EC00032=-798156,1112951
EC00033=-798156,1112951
EC00034=-798156,1112951
EC00035=-798156,1112951
EC00036=-798156,1112951
EC00037=-798156,1112951
EC00038=-798156,1112951
EC00039=-798156,1112951
EC00040=-798156,1112951
EC00041=-798156,1112951
EC00042=-798156,1112951
EC00043=-798156,1112951
EC00044=-798156,1112951
EC00045=-798156,1112951
EC00046=-798156,1112951
EC00047=-798156,1112951
EC00048=-798156,1112951
EC00049=-798156,1112951
EC00050=-798156,1112951
EC00051=-798156,1112951
EC00052=-798156,1112951
EC00053=-798156,1112951
EC00054=-798156,1112951
EC00055=-798156,1112951
EC00056=-798156,1112951
EC00057=-798156,1112951
EC00058=-798156,1112951
EC00059=-798156,1112951
EC00060=-798156,1112951
EC00061=-798156,1112951
EC00062=-798156,1112951
EC00063=-798156,1112951
EC00064=-798156,1112951
EC00065=-798156,1112951
EC00066=-798156,1112951
EC00067=-798156,1112951
EC00068=-798156,1112951
EC00069=-798156,1112951
EC00070=-798156,1112951
EC00071=-798156,1112951
EC00072=-798156,1112951
EC00073=-798156,1112951
EC00074=-798156,1112951
EC00075=-798156,1112951
EC00076=-798156,1112951
EC00077=-798156,1112951
EC00078=-798156,1112951
EC00079=-798156,1112951
EC00080=-798156,1112951
EC00081=-798156,1112951
EC00082=-798156,1112951
EC00083=-798156,1112951
EC00084=-798156,1112951
EC00085=-798156,1112951
EC00086=-798156,1112951
EC00087=-798156,1112951
EC00088=-798156,1112951
EC00089=-798156,1112951
EC00090=-798156,1112951
EC00091=-798156,1112951
EC00092=-798156,1112951
EC00093=-798156,1112951
EC00094=-798156,1112951
EC00095=-798156,1112951
EC00096=-798156,1112951
EC00097=-798156,1112951
EC00098=-798156,1112951
EC00099=-798156,1112951
EC00100=-798156,1112951
EC00101=-798156,1112951
EC00102=-798156,1112951
EC00103=-798156,1112951
EC00104=-798156,1112951
EC00105=-798156,1112951
EC00106=-798156,1112951
EC00107=-798156,1112951
EC00108=-798156,1112951
EC00109=-798156,1112951
EC00110=-798156,1112951
EC00111=-798156,1112951
EC00112=-798156,1112951
EC00113=-798156,1112951
EC00114=-798156,1112951
EC00115=-798156,1112951
EC00116=-798156,1112951
EC00117=-798156,1112951
EC00118=-798156,1112951
EC00119=-798156,1112951
EC00120=-798156,1112951
EC00121=-798156,1112951
EC00122=-798156,1112951
EC00123=-798156,1112951
EC00124=-798156,1112951
EC00125=-798156,1112951
EC00126=-798156,1112951
EC00127=-798156,1112951
EC00128=-798156,1112951
EC00129=-798156,1112951
EC00130=-798156,1112951
EC00131=-798156,1112951
EC00132=-798156,1112951
EC00133=-798156,1112951
EC00134=-798156,1112951
EC00135=-798156,1112951
EC00136=-798156,1112951
EC00137=-798156,1112951
EC00138=-798156,1112951
EC00139=-798156,1112951
EC00140=-798156,1112951
EC00141=-798156,1112951
EC00142=-798156,1112951
EC00143=-798156,1112951
EC00144=-798156,1112951
EC00145=-798156,1112951
EC00146=-798156,1112951
EC00147=-798156,1112951
EC00148=-798156,1112951
EC00149=-798156,1112951
EC00150=-798156,1112951
EC00151=-798156,1112951
EC00152=-798154,1112951
EC00153=-798154,1112951
EC00154=-798156,1112951
EC00155=-798156,1112951
EC00156=-798156,1112951
EC00157=-798156,1112951
EC00158=-798156,1112951
EC00159=-798156,1112951
EC00160=-798156,1112951
EC00161=-798156,1112951
EC00162=-798156,1112951
EC00163=-798156,1112951
EC00164=-798156,1112951
EC00165=-798156,1112951
EC00166=-798156,1112951
EC00167=-798156,1112951
EC00168=-798156,1112951
EC00169=-798156,1112951
EC00170=-798156,1112951
EC00171=-798156,1112951
EC00172=-798156,1112951
EC00173=-798156,1112951
EC00174=-798156,1112951
EC00175=-798156,1112951
EC00176=-798156,1112951
EC00177=-798156,1112951
EC00178=-798156,1112951
EC00179=-798156,1112951
EC00180=-798156,1112951
EC00181=-798156,1112951
EC00182=-798156,1112951
EC00183=-798155,1112952
EC00184=-798155,1112952
EC00185=-798155,1112952
EC00186=-798156,1112951
EC00187=-798156,1112951
EC00188=-798156,1112951
EC00189=-798156,1112951
EC00190=-798156,1112951
EC00191=-798156,1112951
EC00192=-798156,1112951
EC00193=-798155,1112952
EC00194=-798156,1112951
EC00195=-798156,1112951
EC00196=-798156,1112951
EC00197=-798154,1112952
EC00198=-798156,1112951
EC00199=-798156,1112951
EC00200=-798156,1112951
EC00201=-798156,1112951
EC00202=-798156,1112951
EC00203=-798156,1112951
EC00204=-798156,1112951
EC00205=-798156,1112951
EC00206=-798156,1112951
EC00207=-798156,1112951
EC00208=-798156,1112951
EC00209=-798156,1112951
EC00210=-798156,1112951
EC00211=-798156,1112951
EC00212=-798156,1112951
EC00213=-798156,1112951
EC00214=-798156,1112951
EC00215=-798156,1112951
EC00216=-798156,1112951
EC00217=-798156,1112951
EC00218=-798156,1112951
EC00219=-798156,1112951
EC00220=-798156,1112951
EC00221=-798156,1112951
EC00222=-798156,1112951
EC00223=-798156,1112951
EC00224=-798156,1112951
EC00225=-798156,1112951
EC00226=-798156,1112951
EC00227=-798156,1112951
EC00228=-798155,1112952
EC00229=-798155,1112952
EC00230=-798155,1112952
EC00231=-798156,1112951
EC00232=-798156,1112951
EC00233=-798156,1112951
EC00234=-798156,1112951
EC00235=-798156,1112951
EC00236=-798156,1112951
EC00237=-798156,1112951
EC00238=-798156,1112951
EC00239=-798156,1112951
EC00240=-798156,1112951
EC00241=-798156,1112951
EC00242=-798156,1112951
EC00243=-798156,1112951
EC00244=-798156,1112951
EC00245=-798156,1112951
EC00246=-798156,1112951
EC00247=-888531,899777
EC00248=-888287,769744
EC00249=-887396,295576
EC00250=-886840,0
EC00251=-798156,0
EC00252=-798156,0
EC00253=-798156,0
EC00254=-798156,0
EC00255=-798156,0
EC00256=-798156,0
EC00257=-798156,0
EC00258=-798156,0
EC00259=-798156,0
EC00260=-798156,0
EC00261=-798156,0
EC00262=-798156,0
EC00263=-798156,0
EC00264=-798156,0
EC00265=-798156,0
EC00266=-798156,0
EC00267=-798156,0
EC00268=-798156,0
EC00269=-798156,0
EC00270=-798156,0
EC00271=-798156,0
EC00272=-798156,0
EC00273=-798156,0
EC00274=-798156,0
EC00275=-798156,0
EC00276=-798156,0
EC00277=-798156,0
EC00278=-798156,0
EC00279=-798156,0
EC00280=-798156,0
EC00281=-798156,0
EC00282=-798156,0
EC00283=-798156,0
EC00284=-798156,0
EC00285=-798156,0
EC00286=-798156,0
EC00287=-798156,0
EC00288=-798156,0
EC00289=-798156,0
EC00290=-798156,0
EC00291=-798156,0
EC00292=-798156,0
EC00293=-798156,0
EC00294=-798156,0
EC00295=-798156,0
EC00296=-798156,0
EC00297=-798156,0
EC00298=-798156,0
EC00299=-798156,0
EC00300=-798156,0
EC00301=-798156,0
EC00302=-798156,0
EC00303=-798156,0
EC00304=-798156,0
EC00305=-798156,0
EC00306=-798156,0
EC00307=-798156,0
EC00308=-798156,0
EC00309=-798156,0
EC00310=-798156,0
EC00311=-798156,0
EC00312=-798156,0
EC00313=-798156,0
EC00314=-798156,0
EC00315=-798156,0
EC00316=-798154,0
EC00317=-798154,0
EC00318=-798154,0
EC00319=-798154,0
EC00320=-798154,0
EC00321=-798154,0
EC00322=-798156,0
EC00323=-798156,0
EC00324=-798156,0
EC00325=-798156,0
EC00326=-798156,0
EC00327=-798156,0
EC00328=-798156,0
EC00329=-798156,0
EC00330=-798156,0
EC00331=-798156,0
EC00332=-798156,0
EC00333=-798156,0
EC00334=-798156,0
EC00335=-798156,0
EC00336=-798156,0
EC00337=-798156,0
EC00338=-798156,0
EC00339=-798156,0
EC00340=-798156,0
EC00341=-798156,0
EC00342=-798156,0
EC00343=-798156,0
EC00344=-798156,0
EC00345=-798156,0
EC00346=-798156,0
EC00347=-798156,0
EC00348=-798156,0
EC00349=-798156,0
EC00350=-798156,0
EC00351=-798156,0
EC00352=-798156,0
EC00353=-798156,0
EC00354=-798156,0
EC00355=-798156,0
EC00356=-798156,0
EC00357=-798156,0
EC00358=-798156,0
EC00359=-798156,0
EC00360=-798156,0
EC00361=-798156,0
EC00362=-798156,0
EC00363=-798156,0
EC00364=-798156,0
EC00365=-798156,0
EC00366=-798156,0
EC00367=-798156,0
EC00368=-798156,0
EC00369=-798156,0
EC00370=-798156,0
EC00371=-798156,0
EC00372=-798156,0
EC00373=-798156,0
EC00374=-798156,0
EC00375=-798156,0
EC00376=-798156,0
EC00377=-798156,0
EC00378=-798156,0
EC00379=-798156,0
EC00380=-798156,0
EC00381=-798156,0
EC00382=-798156,0
EC00383=-798156,0
EC00384=-798156,0
EC00385=-798156,0
EC00386=-798156,0
EC00387=-798156,0
EC00388=-798156,0
EC00389=-798156,0
EC00390=-798156,0
EC00391=-798156,0
EC00392=-798156,0
EC00393=-798156,0
EC00394=-798156,0
EC00395=-798156,0
EC00396=-798156,0
EC00397=-798156,0
EC00398=-798156,0
EC00399=-798156,0
EC00400=-798156,0
EC00401=-798156,0
EC00402=-798156,0
EC00403=-798156,0
EC00404=-798156,0
EC00405=-798156,0
EC00406=-798156,0
EC00407=-798156,0
EC00408=-798156,0
EC00409=-798156,0
EC00410=-798156,0
EC00411=-798156,0
EC00412=-798151,0
EC00413=-798156,0
EC00414=-798156,0
EC00415=-798152,0
EC00416=-798152,0
EC00417=-798152,0
EC00418=-798152,0
EC00419=-798152,0
EC00420=-798156,0
EC00421=-798156,0
EC00422=-798156,0
EC00423=-798156,0
EC00424=-798156,0
EC00425=-798156,0
EC00426=-798156,0
EC00427=-798156,0
EC00428=-798156,0
EC00429=-798156,0
EC00430=-798156,0
EC00431=-798156,0
EC00432=-798156,0
EC00433=-798156,0
EC00434=-798156,0
EC00435=-798156,0
EC00436=-798156,0
EC00437=-798156,0
EC00438=-798156,0
EC00439=-798156,0
EC00440=-798156,0
EC00441=-798156,0
EC00442=-798156,0
EC00443=-798156,0
EC00444=-798156,0
EC00445=-798156,0
EC00446=-798156,0
EC00447=-798156,0
EC00448=-798156,0
EC00449=-798156,0
EC00450=-798156,0
EC00451=-798156,0
EC00452=-798156,0
EC00453=-798156,0
EC00454=-798156,0
EC00455=-798156,0
EC00456=-798156,0
EC00457=-798156,0
EC00458=-798156,0
EC00459=-798156,0
EC00460=-798156,0
EC00461=-798156,0
EC00462=-798156,0
EC00463=-798156,0
EC00464=-798156,0
EC00465=-798156,0
EC00466=-798156,0
EC00467=-798156,0
EC00468=-798156,0
EC00469=-798155,-1
EC00470=-798156,0
EC00471=-798156,0
EC00472=-798155,-1
EC00473=-798156,0
EC00474=-798156,0
EC00475=-798156,0
EC00476=-798156,0
EC00477=-798156,0
EC00478=-798156,0
EC00479=-805602,0
EC00480=-805602,0
///POSTYPE BASE
///RECTAN
///RCONF 0,0,0,0,0,0,0,0,0,0,0,0,0,0,0,0,0,0,0,0,0,0,0,0
P00006=0.222,-3.123,-1.508,0.0000,0.0000,0.0000
P00021=-0.225,-6.128,-0.405,0.0000,0.0000,0.0000
P00022=0.222,-3.123,-1.508,0.0000,0.0000,0.0000
P00023=0.143,-0.036,0.682,0.0000,0.0000,0.0000
P00024=0.145,-0.552,1.326,0.0000,0.0000,0.0000
P00031=1.853,-0.001,-1.549,0.0000,0.0000,0.0000
P00032=1.957,0.503,-7.217,0.0000,0.0000,0.0000
///RCONF 0,0,0,0,1,0,0,0,0,0,0,0,0,0,0,0,0,0,0,0,0,0,0,0
P00033=-0.123,0.612,-5.012,0.0000,0.0000,0.0000
///RCONF 0,0,0,0,0,0,0,0,0,0,0,0,0,0,0,0,0,0,0,0,0,0,0,0
P00035=2.817,0.591,-1.622,0.0000,0.0000,0.0000
P00036=-1.108,-0.829,1.850,0.0000,0.0000,0.0000
P00037=0.023,0.937,-2.677,0.0000,0.0000,0.0000
P00038=0.158,-1.133,-1.952,0.0000,0.0000,0.0000
P00039=0.012,-3.081,-0.106,0.0000,0.0000,0.0000
P00040=-0.030,9.648,2.467,0.0000,0.0000,0.0000
P00050=4.296,-4.501,-0.826,0.0000,0.0000,0.0000
P00051=0.367,3.892,0.009,0.0000,0.0000,0.0000
P00052=0.088,2.832,-0.342,0.0000,0.0000,0.0000
P00053=0.134,6.594,0.107,0.0000,0.0000,0.0000
P00054=-0.103,6.509,-0.702,0.0000,0.0000,0.0000
P00059=0.483,-0.984,-2.888,0.0000,0.0000,0.0000
P00060=2.327,-2.514,-2.692,0.0000,0.0000,0.0000
P00061=1.575,-3.405,-0.752,0.0000,0.0000,0.0000
P00062=-0.135,-0.848,-1.706,0.0000,0.0000,0.0000
P00070=0.003,2.805,-1.116,0.0000,0.0000,0.0000
P00071=2.716,0.070,1.352,0.0000,0.0000,0.0000
P00072=1.041,-0.003,-0.797,0.0000,0.0000,0.0000
P00073=-0.961,5.319,-6.157,0.0000,0.0000,0.0000
P00074=1.123,1.944,-5.914,0.0000,0.0000,0.0000
///RCONF 0,1,0,0,0,0,0,0,0,0,0,0,0,0,0,0,0,0,0,0,0,0,0,0
P00075=-1.802,0.025,1.546,0.0000,0.0000,0.0000
//INST
///DATE 2025/01/22 12:53
///ATTR SC,RW
///GROUP1 RB1,BS1
///GROUP2 ST1
NOP
'OK_r2_O29-32(90,0_180)
'-90,180
'Path S1470
SFTOF3D
MOVJ C00000 BC00000 VJ=100.00  +MOVJ EC00000 VJ=100.00
MOVJ C00001 BC00001 VJ=100.00  +MOVJ EC00001 VJ=100.00
SMOVL C00002 BC00002 V=500.0  +MOVJ EC00002
SMOVL C00003 BC00003 V=166.7  +MOVJ EC00003
SREFP 3 C00004 BC00004  +REFP EC00004
CALL JOB:SEARCH-R1-S13D
SET P059 P006
SFTON3D P059
SMOVL C00005 BC00005 V=166.7  +MOVJ EC00005
SREFP 3 C00006 BC00006  +REFP EC00006
CALL JOB:SEARCH-R1-S13D
SET P059 P006
SFTON3D P059
SMOVL C00007 BC00007 V=166.7  +MOVJ EC00007
SFTOF3D
MOVL C00008 BC00008 V=250.0  +MOVJ EC00008 VJ=100.00
SREFP 3 C00009 BC00009  +REFP EC00009
CALL JOB:SEARCH-R1-S13D
SET P021 P006
SFTON3D P021
SMOVL C00010 BC00010 V=166.7  +MOVJ EC00010
SREFP 3 C00011 BC00011  +REFP EC00011
CALL JOB:SEARCH-R1-S13D
SET P021 P006
SFTON3D P021
SMOVL C00012 BC00012 V=166.7  +MOVJ EC00012
SREFP 3 C00013 BC00013  +REFP EC00013
CALL JOB:SEARCH-R1-S13D
SET P021 P006
SFTON3D P021
SMOVL C00014 BC00014 V=166.7  +MOVJ EC00014
SFTOF3D
MOVL C00015 BC00015 V=400.0  +MOVJ EC00015 VJ=100.00
MOVL C00016 BC00016 V=1000.0  +MOVJ EC00016 VJ=100.00
MOVJ C00017 BC00017 VJ=100.00  +MOVJ EC00017 VJ=100.00
MOVL C00018 BC00018 V=166.7  +MOVJ EC00018 VJ=100.00
SMOVL C00019 BC00019 V=166.7  +MOVJ EC00019
SREFP 3 C00020 BC00020  +REFP EC00020
CALL JOB:SEARCH-R1-S13D
SET P022 P006
SFTON3D P022
SMOVL C00021 BC00021 V=166.7  +MOVJ EC00021
SREFP 3 C00022 BC00022  +REFP EC00022
CALL JOB:SEARCH-R1-S13D
SET P022 P006
SFTON3D P022
SMOVL C00023 BC00023 V=166.7  +MOVJ EC00023
SMOVL C00024 BC00024 V=250.0  +MOVJ EC00024
SMOVL C00025 BC00025 V=166.7  +MOVJ EC00025
SREFP 3 C00026 BC00026  +REFP EC00026
CALL JOB:SEARCH-R1-S13D
SET P022 P006
SFTON3D P022
SMOVL C00027 BC00027 V=250.0  +MOVJ EC00027
MOVL C00028 BC00028 V=1000.0  +MOVJ EC00028 VJ=100.00
'Path S1472
SFTOF3D
MOVJ C00029 BC00029 VJ=100.00  +MOVJ EC00029 VJ=20.00
MOVJ C00030 BC00030 VJ=100.00  +MOVJ EC00030 VJ=100.00
MOVL C00031 BC00031 V=400.0  +MOVJ EC00031 VJ=100.00
SMOVL C00032 BC00032 V=166.7  +MOVJ EC00032
SREFP 3 C00033 BC00033  +REFP EC00033
CALL JOB:SEARCH-R1-S13D
SET P023 P006
SFTON3D P023
SMOVL C00034 BC00034 V=166.7  +MOVJ EC00034
SMOVL C00035 BC00035 V=166.7  +MOVJ EC00035
SMOVL C00036 BC00036 V=166.7  +MOVJ EC00036
SREFP 3 C00037 BC00037  +REFP EC00037
CALL JOB:SEARCH-R1-S13D
SET P023 P006
SFTON3D P023
SMOVL C00038 BC00038 V=166.7  +MOVJ EC00038
SMOVL C00039 BC00039 V=250.0  +MOVJ EC00039
SMOVL C00040 BC00040 V=250.0  +MOVJ EC00040
SREFP 3 C00041 BC00041  +REFP EC00041
CALL JOB:SEARCH-R1-S13D
SET P023 P006
SFTON3D P023
SMOVL C00042 BC00042 V=250.0  +MOVJ EC00042
MOVL C00043 BC00043 V=250.0  +MOVJ EC00043 VJ=100.00
MOVL C00044 BC00044 V=500.0  +MOVJ EC00044 VJ=100.00
'Path S1473
SFTOF3D
MOVJ C00045 BC00045 VJ=40.00  +MOVJ EC00045 VJ=100.00
MOVL C00046 BC00046 V=400.0  +MOVJ EC00046 VJ=100.00
SMOVL C00047 BC00047 V=166.7  +MOVJ EC00047
SREFP 3 C00048 BC00048  +REFP EC00048
CALL JOB:SEARCH-R1-S13D
SET P024 P006
SFTON3D P024
SMOVL C00049 BC00049 V=166.7  +MOVJ EC00049
SREFP 3 C00050 BC00050  +REFP EC00050
CALL JOB:SEARCH-R1-S13D
SET P024 P006
SFTON3D P024
SMOVL C00051 BC00051 V=166.7  +MOVJ EC00051
SFTOF3D
MOVL C00052 BC00052 V=400.0  +MOVJ EC00052 VJ=100.00
SMOVL C00053 BC00053 V=666.7  +MOVJ EC00053
SMOVL C00054 BC00054 V=166.7  +MOVJ EC00054
SREFP 3 C00055 BC00055  +REFP EC00055
CALL JOB:SEARCH-R1-S13D
SET P060 P006
SFTON3D P060
SMOVL C00056 BC00056 V=166.7  +MOVJ EC00056
SREFP 3 C00057 BC00057  +REFP EC00057
CALL JOB:SEARCH-R1-S13D
SET P060 P006
SFTON3D P060
SMOVL C00058 BC00058 V=166.7  +MOVJ EC00058
SFTOF3D
SMOVL C00059 BC00059 V=500.0  +MOVJ EC00059
SMOVL C00060 BC00060 V=166.7  +MOVJ EC00060
SREFP 3 C00061 BC00061  +REFP EC00061
CALL JOB:SEARCH-R1-S13D
SET P061 P006
SFTON3D P061
SMOVL C00062 BC00062 V=166.7  +MOVJ EC00062
SREFP 3 C00063 BC00063  +REFP EC00063
CALL JOB:SEARCH-R1-S13D
SET P061 P006
SFTON3D P061
SMOVL C00064 BC00064 V=166.7  +MOVJ EC00064
MOVL C00065 BC00065 V=1000.0  +MOVJ EC00065 VJ=100.00
'Path S1466
SFTOF3D
MOVJ C00066 BC00066 VJ=100.00  +MOVJ EC00066 VJ=100.00
MOVL C00067 BC00067 V=400.0  +MOVJ EC00067 VJ=100.00
SMOVL C00068 BC00068 V=100.0  +MOVJ EC00068
SREFP 3 C00069 BC00069  +REFP EC00069
CALL JOB:SEARCH-R1-S13D
SET P038 P006
SFTON3D P038
SMOVL C00070 BC00070 V=100.0  +MOVJ EC00070
SREFP 3 C00071 BC00071  +REFP EC00071
CALL JOB:SEARCH-R1-S13D
SET P038 P006
SFTON3D P038
SMOVL C00072 BC00072 V=100.0  +MOVJ EC00072
SFTOF3D
SMOVL C00073 BC00073 V=666.7  +MOVJ EC00073
SMOVL C00074 BC00074 V=166.7  +MOVJ EC00074
SREFP 3 C00075 BC00075  +REFP EC00075
CALL JOB:SEARCH-R1-S13D
SET P062 P006
SFTON3D P062
SMOVL C00076 BC00076 V=166.7  +MOVJ EC00076
SREFP 3 C00077 BC00077  +REFP EC00077
CALL JOB:SEARCH-R1-S13D
SET P062 P006
SFTON3D P062
SMOVL C00078 BC00078 V=166.7  +MOVJ EC00078
MOVL C00079 BC00079 V=1000.0  +MOVJ EC00079 VJ=100.00
SFTOF3D
MOVJ C00080 BC00080 VJ=100.00  +MOVJ EC00080 VJ=100.00
MOVJ C00081 BC00081 VJ=100.00  +MOVJ EC00081 VJ=100.00
MOVJ C00082 BC00082 VJ=100.00  +MOVJ EC00082 VJ=20.00
MOVJ C00083 BC00083 VJ=100.00  +MOVJ EC00083 VJ=100.00
MOVJ C00084 BC00084 VJ=100.00  +MOVJ EC00084 VJ=100.00
MOVJ C00085 BC00085 VJ=100.00  +MOVJ EC00085 VJ=100.00
MOVJ C00086 BC00086 VJ=100.00  +MOVJ EC00086 VJ=100.00
MOVJ C00087 BC00087 VJ=100.00  +MOVJ EC00087 VJ=100.00
'Path S1047
SMOVL C00088 BC00088 V=166.7  +MOVJ EC00088
SREFP 3 C00089 BC00089  +REFP EC00089
CALL JOB:SEARCH-R1-S13D
SET P071 P006
SFTON3D P071
SMOVL C00090 BC00090 V=166.7  +MOVJ EC00090
SMOVL C00091 BC00091 V=166.7  +MOVJ EC00091
SMOVL C00092 BC00092 V=166.7  +MOVJ EC00092
SREFP 3 C00093 BC00093  +REFP EC00093
CALL JOB:SEARCH-R1-S13D
SET P071 P006
SFTON3D P071
SMOVL C00094 BC00094 V=166.7  +MOVJ EC00094
SMOVL C00095 BC00095 V=666.7  +MOVJ EC00095
SMOVL C00096 BC00096 V=166.7  +MOVJ EC00096
SREFP 3 C00097 BC00097  +REFP EC00097
CALL JOB:SEARCH-R1-S13D
SET P072 P006
SFTON3D P072
SMOVL C00098 BC00098 V=166.7  +MOVJ EC00098
SMOVL C00099 BC00099 V=166.7  +MOVJ EC00099
SMOVL C00100 BC00100 V=166.7  +MOVJ EC00100
SREFP 3 C00101 BC00101  +REFP EC00101
CALL JOB:SEARCH-R1-S13D
SET P072 P006
SFTON3D P072
SMOVL C00102 BC00102 V=166.7  +MOVJ EC00102
SMOVL C00103 BC00103 V=166.7  +MOVJ EC00103
SREFP 3 C00104 BC00104  +REFP EC00104
CALL JOB:SEARCH-R1-S13D
SET P073 P006
SFTON3D P073
SMOVL C00105 BC00105 V=166.7  +MOVJ EC00105
SMOVL C00106 BC00106 V=166.7  +MOVJ EC00106
SMOVL C00107 BC00107 V=166.7  +MOVJ EC00107
SREFP 3 C00108 BC00108  +REFP EC00108
CALL JOB:SEARCH-R1-S13D
SET P073 P006
SFTON3D P073
SMOVL C00109 BC00109 V=166.7  +MOVJ EC00109
SMOVL C00110 BC00110 V=666.7  +MOVJ EC00110
SMOVL C00111 BC00111 V=166.7  +MOVJ EC00111
SREFP 3 C00112 BC00112  +REFP EC00112
CALL JOB:SEARCH-R1-S13D
SET P074 P006
SFTON3D P074
SMOVL C00113 BC00113 V=166.7  +MOVJ EC00113
SMOVL C00114 BC00114 V=166.7  +MOVJ EC00114
SMOVL C00115 BC00115 V=166.7  +MOVJ EC00115
SREFP 3 C00116 BC00116  +REFP EC00116
CALL JOB:SEARCH-R1-S13D
SET P074 P006
SFTON3D P074
SMOVL C00117 BC00117 V=166.7  +MOVJ EC00117
SMOVL C00118 BC00118 V=166.7  +MOVJ EC00118
SMOVL C00119 BC00119 V=166.7  +MOVJ EC00119
SREFP 3 C00120 BC00120  +REFP EC00120
CALL JOB:SEARCH-R1-S13D
SET P075 P006
SFTON3D P075
SMOVL C00121 BC00121 V=166.7  +MOVJ EC00121
SMOVL C00122 BC00122 V=166.7  +MOVJ EC00122
SMOVL C00123 BC00123 V=166.7  +MOVJ EC00123
SREFP 3 C00124 BC00124  +REFP EC00124
CALL JOB:SEARCH-R1-S13D
SET P075 P006
SFTON3D P075
SMOVL C00125 BC00125 V=166.7  +MOVJ EC00125
SFTOF3D
SMOVL C00126 BC00126 V=666.7  +MOVJ EC00126
SMOVL C00127 BC00127 V=666.7  +MOVJ EC00127
MOVJ C00128 BC00128 VJ=100.00  +MOVJ EC00128 VJ=100.00
MOVL C00129 BC00129 V=400.0  +MOVJ EC00129 VJ=100.00
SMOVL C00130 BC00130 V=166.7  +MOVJ EC00130
SREFP 3 C00131 BC00131  +REFP EC00131
CALL JOB:SEARCH-R1-S13D
SET P031 P006
SFTON3D P031
SMOVL C00132 BC00132 V=166.7  +MOVJ EC00132
SMOVL C00133 BC00133 V=166.7  +MOVJ EC00133
SREFP 3 C00134 BC00134  +REFP EC00134
CALL JOB:SEARCH-R1-S13D
SET P031 P006
SFTON3D P031
SMOVL C00135 BC00135 V=166.7  +MOVJ EC00135
MOVL C00136 BC00136 V=400.0  +MOVJ EC00136 VJ=100.00
MOVJ C00137 BC00137 VJ=100.00  +MOVJ EC00137 VJ=100.00
'KAT_ZMIANA
MOVJ C00138 BC00138 VJ=100.00  +MOVJ EC00138 VJ=20.00
'-90,180
'Path W1014
SFTOF3D
SMOVL C00139 BC00139 V=400.0  +MOVJ EC00139
SMOVL C00140 BC00140 V=333.3  +MOVJ EC00140
SMOVL C00141 BC00141 V=100.0  +MOVJ EC00141
SREFP 3 C00142 BC00142  +REFP EC00142
CALL JOB:SEARCH-R1-S13D
SET P040 P006
SFTON3D P040
SMOVL C00143 BC00143 V=100.0  +MOVJ EC00143
SREFP 3 C00144 BC00144  +REFP EC00144
CALL JOB:SEARCH-R1-S13D
SET P040 P006
SFTON3D P040
SMOVL C00145 BC00145 V=166.7  +MOVJ EC00145
SMOVL C00146 BC00146 V=400.0  +MOVJ EC00146
SFTON3D P031
SMOVL C00147 BC00147 V=166.7 PL=0  +MOVJ EC00147
SREFP 1 C00148 BC00148  +REFP EC00148
SREFP 2 C00149 BC00149  +REFP EC00149
MACRO1 MJ#(0) ARGF14
ARCON
SMOVL C00150 BC00150 V=8.3  +MOVJ EC00150
SFTON3D P040
SMOVL C00151 BC00151 V=8.3  +MOVJ EC00151
SMOVL C00152 BC00152 V=8.3  +MOVJ EC00152
ARCOF
SMOVL C00153 BC00153 V=400.0  +MOVJ EC00153
SFTOF3D
MOVJ C00154 BC00154 VJ=100.00  +MOVJ EC00154 VJ=100.00
SMOVL C00155 BC00155 V=666.7  +MOVJ EC00155
SFTON3D P075
SMOVL C00156 BC00156 V=666.7  +MOVJ EC00156
SMOVL C00157 BC00157 V=666.7  +MOVJ EC00157
SMOVL C00158 BC00158 V=166.7 PL=0  +MOVJ EC00158
MACRO1 MJ#(0) ARGF9
ARCON
SMOVL C00159 BC00159 V=13.3  +MOVJ EC00159
SMOVC C00160 BC00160 V=15.0  +MOVJ EC00160
SMOVC C00161 BC00161 V=15.0  +MOVJ EC00161
SMOVC C00162 BC00162 V=15.0  +MOVJ EC00162
SMOVL C00163 BC00163 V=12.5  +MOVJ EC00163
SFTON3D P074
SMOVL C00164 BC00164 V=12.5  +MOVJ EC00164
SMOVC C00165 BC00165 V=15.0  +MOVJ EC00165
SMOVC C00166 BC00166 V=15.0  +MOVJ EC00166
SFTON3D P073
SMOVC C00167 BC00167 V=15.0  +MOVJ EC00167
SFTON3D P072
SMOVL C00168 BC00168 V=12.5  +MOVJ EC00168
ARCOF
SMOVL C00169 BC00169 V=166.7  +MOVJ EC00169
SFTOF3D
SMOVL C00170 BC00170 V=666.7  +MOVJ EC00170
SMOVL C00171 BC00171 V=666.7  +MOVJ EC00171
MOVJ C00172 BC00172 VJ=100.00  +MOVJ EC00172 VJ=100.00
MOVJ C00173 BC00173 VJ=100.00  +MOVJ EC00173 VJ=100.00
MOVJ C00174 BC00174 VJ=100.00  +MOVJ EC00174 VJ=20.00
MOVJ C00175 BC00175 VJ=100.00  +MOVJ EC00175 VJ=100.00
MOVJ C00176 BC00176 VJ=100.00  +MOVJ EC00176 VJ=100.00
MOVJ C00177 BC00177 VJ=100.00  +MOVJ EC00177 VJ=100.00
'Path W1467
SFTOF3D
SFTON3D P038
MOVJ C00178 BC00178 VJ=100.00  +MOVJ EC00178 VJ=100.00
SMOVL C00179 BC00179 V=400.0  +MOVJ EC00179
SMOVL C00180 BC00180 V=133.3 PL=0  +MOVJ EC00180
SREFP 1 C00181 BC00181  +REFP EC00181
SREFP 2 C00182 BC00182  +REFP EC00182
MACRO1 MJ#(0) ARGF6
ARCON
SMOVL C00183 BC00183 V=8.3  +MOVJ EC00183
SFTON3D P062
SMOVL C00184 BC00184 V=8.3  +MOVJ EC00184
SMOVL C00185 BC00185 V=8.3  +MOVJ EC00185
ARCOF
SMOVL C00186 BC00186 V=400.0  +MOVJ EC00186
SFTOF3D
'Path W1473
SFTOF3D
SFTON3D P061
MOVJ C00187 BC00187 VJ=100.00  +MOVJ EC00187 VJ=20.00
MOVJ C00188 BC00188 VJ=100.00  +MOVJ EC00188 VJ=100.00
SMOVL C00189 BC00189 V=400.0  +MOVJ EC00189
SMOVL C00190 BC00190 V=133.3 PL=0  +MOVJ EC00190
SREFP 1 C00191 BC00191  +REFP EC00191
SREFP 2 C00192 BC00192  +REFP EC00192
MACRO1 MJ#(0) ARGF14
ARCON
SFTON3D P022
SMOVL C00193 BC00193 V=8.3  +MOVJ EC00193
ARCOF
SMOVL C00194 BC00194 V=333.3  +MOVJ EC00194
SFTOF3D
SFTOF3D
'Path W1474
SFTOF3D
MOVJ C00195 BC00195 VJ=15.00  +MOVJ EC00195 VJ=100.00
MOVJ C00196 BC00196 VJ=15.00  +MOVJ EC00196 VJ=100.00
SFTON3D P059
SMOVL C00197 BC00197 V=133.3 PL=0  +MOVJ EC00197
SREFP 1 C00198 BC00198  +REFP EC00198
SREFP 2 C00199 BC00199  +REFP EC00199
MACRO1 MJ#(0) ARGF14
ARCON
SFTON3D P021
SMOVL C00200 BC00200 V=8.3  +MOVJ EC00200
SMOVL C00201 BC00201 V=8.3  +MOVJ EC00201
SMOVL C00202 BC00202 V=8.3  +MOVJ EC00202
ARCOF
SMOVL C00203 BC00203 V=400.0  +MOVJ EC00203
SMOVL C00204 BC00204 V=1000.0  +MOVJ EC00204
SFTOF3D
'Path W1475
SFTOF3D
SFTON3D P023
SMOVL C00205 BC00205 V=250.0  +MOVJ EC00205
SMOVL C00206 BC00206 V=166.7  +MOVJ EC00206
SREFP 1 C00207 BC00207  +REFP EC00207
SREFP 2 C00208 BC00208  +REFP EC00208
MACRO1 MJ#(0) ARGF14
ARCON
SMOVL C00209 BC00209 V=8.3  +MOVJ EC00209
SFTON3D P021
SMOVL C00210 BC00210 V=8.3  +MOVJ EC00210
SMOVL C00211 BC00211 V=8.3  +MOVJ EC00211
ARCOF
SMOVL C00212 BC00212 V=400.0  +MOVJ EC00212
SMOVL C00213 BC00213 V=1000.0  +MOVJ EC00213
SMOVL C00214 BC00214 V=1000.0  +MOVJ EC00214
SFTOF3D
'Path W1476
SFTOF3D
SFTON3D P023
SMOVL C00215 BC00215 V=166.7  +MOVJ EC00215
SMOVL C00216 BC00216 V=100.0 PL=0  +MOVJ EC00216
SREFP 1 C00217 BC00217  +REFP EC00217
SREFP 2 C00218 BC00218  +REFP EC00218
MACRO1 MJ#(0) ARGF6
ARCON
SMOVL C00219 BC00219 V=12.5  +MOVJ EC00219
ARCOF
SMOVL C00220 BC00220 V=400.0  +MOVJ EC00220
SMOVL C00221 BC00221 V=1000.0  +MOVJ EC00221
SFTOF3D
'Path W1477
SFTOF3D
SFTON3D P024
MOVJ C00222 BC00222 VJ=100.00  +MOVJ EC00222 VJ=100.00
SMOVL C00223 BC00223 V=166.7  +MOVJ EC00223
SMOVL C00224 BC00224 V=166.7 PL=0  +MOVJ EC00224
SREFP 1 C00225 BC00225  +REFP EC00225
SREFP 2 C00226 BC00226  +REFP EC00226
MACRO1 MJ#(0) ARGF14
ARCON
SMOVL C00227 BC00227 V=8.3  +MOVJ EC00227
SMOVL C00228 BC00228 V=8.3  +MOVJ EC00228
ARCOF
SMOVL C00229 BC00229 V=8.3  +MOVJ EC00229
ARCON
SMOVL C00230 BC00230 V=8.3  +MOVJ EC00230
SFTON3D P060
SMOVL C00231 BC00231 V=8.3  +MOVJ EC00231
SMOVL C00232 BC00232 V=8.3  +MOVJ EC00232
ARCOF
SMOVL C00233 BC00233 V=400.0  +MOVJ EC00233
MOVJ C00234 BC00234 VJ=100.00  +MOVJ EC00234 VJ=20.00
SFTOF3D
'Path W1478
SFTOF3D
SFTON3D P022
MOVJ C00235 BC00235 VJ=100.00  +MOVJ EC00235 VJ=100.00
SMOVL C00236 BC00236 V=333.3  +MOVJ EC00236
SMOVL C00237 BC00237 V=133.3 PL=0  +MOVJ EC00237
SREFP 1 C00238 BC00238  +REFP EC00238
SREFP 2 C00239 BC00239  +REFP EC00239
MACRO1 MJ#(0) ARGF6
ARCON
SMOVL C00240 BC00240 V=12.5  +MOVJ EC00240
SMOVL C00241 BC00241 V=12.5  +MOVJ EC00241
ARCOF
SMOVL C00242 BC00242 V=250.0  +MOVJ EC00242
SMOVL C00243 BC00243 V=1000.0  +MOVJ EC00243
MOVJ C00244 BC00244 VJ=100.00  +MOVJ EC00244 VJ=20.00
MOVJ C00245 BC00245 VJ=100.00  +MOVJ EC00245 VJ=20.00
MOVJ C00246 BC00246 VJ=100.00  +MOVJ EC00246 VJ=20.00
CALL JOB:CLEAN-R1_KM_NEW
SFTOF3D
'KAT_ZMIANA
MOVJ C00247 BC00247 VJ=100.00  +MOVJ EC00247 VJ=20.00
MOVJ C00248 BC00248 VJ=100.00  +MOVJ EC00248 VJ=100.00
MOVJ C00249 BC00249 VJ=100.00  +MOVJ EC00249 VJ=100.00
MOVJ C00250 BC00250 VJ=100.00  +MOVJ EC00250 VJ=100.00
MOVJ C00251 BC00251 VJ=100.00  +MOVJ EC00251 VJ=100.00
'-90,0
MOVJ C00252 BC00252 VJ=100.00  +MOVJ EC00252 VJ=100.00
MOVJ C00253 BC00253 VJ=100.00  +MOVJ EC00253 VJ=100.00
'Path S1464
SFTOF3D
MOVJ C00254 BC00254 VJ=100.00  +MOVJ EC00254 VJ=100.00
MOVL C00255 BC00255 V=166.7  +MOVJ EC00255 VJ=100.00
SMOVL C00256 BC00256 V=100.0  +MOVJ EC00256
SREFP 3 C00257 BC00257  +REFP EC00257
CALL JOB:SEARCH-R1-S13D
SET P037 P006
SFTON3D P037
SMOVL C00258 BC00258 V=100.0  +MOVJ EC00258
SMOVL C00259 BC00259 V=100.0  +MOVJ EC00259
SREFP 3 C00260 BC00260  +REFP EC00260
CALL JOB:SEARCH-R1-S13D
SET P037 P006
SFTON3D P037
SMOVL C00261 BC00261 V=100.0  +MOVJ EC00261
SFTOF3D
MOVL C00262 BC00262 V=400.0  +MOVJ EC00262 VJ=100.00
SMOVL C00263 BC00263 V=250.0  +MOVJ EC00263
SMOVL C00264 BC00264 V=100.0  +MOVJ EC00264
SREFP 3 C00265 BC00265  +REFP EC00265
CALL JOB:SEARCH-R1-S13D
SET P050 P006
SFTON3D P050
SMOVL C00266 BC00266 V=100.0  +MOVJ EC00266
SREFP 3 C00267 BC00267  +REFP EC00267
CALL JOB:SEARCH-R1-S13D
SET P050 P006
SFTON3D P050
SMOVL C00268 BC00268 V=100.0  +MOVJ EC00268
SMOVL C00269 BC00269 V=250.0  +MOVJ EC00269
MOVL C00270 BC00270 V=1000.0  +MOVJ EC00270 VJ=100.00
MOVJ C00271 BC00271 VJ=100.00  +MOVJ EC00271 VJ=100.00
MOVJ C00272 BC00272 VJ=100.00  +MOVJ EC00272 VJ=100.00
MOVJ C00273 BC00273 VJ=100.00  +MOVJ EC00273 VJ=100.00
MOVJ C00274 BC00274 VJ=100.00  +MOVJ EC00274 VJ=100.00
'Path S1468
SFTOF3D
MOVJ C00275 BC00275 VJ=100.00  +MOVJ EC00275 VJ=100.00
MOVL C00276 BC00276 V=250.0  +MOVJ EC00276 VJ=100.00
SMOVL C00277 BC00277 V=166.7  +MOVJ EC00277
SREFP 3 C00278 BC00278  +REFP EC00278
CALL JOB:SEARCH-R1-S13D
SET P039 P006
SFTON3D P039
SMOVL C00279 BC00279 V=100.0  +MOVJ EC00279
SMOVL C00280 BC00280 V=100.0  +MOVJ EC00280
SREFP 3 C00281 BC00281  +REFP EC00281
CALL JOB:SEARCH-R1-S13D
SET P039 P006
SFTON3D P039
SMOVL C00282 BC00282 V=100.0  +MOVJ EC00282
SFTOF3D
MOVL C00283 BC00283 V=400.0  +MOVJ EC00283 VJ=100.00
SMOVL C00284 BC00284 V=333.3  +MOVJ EC00284
SMOVL C00285 BC00285 V=250.0  +MOVJ EC00285
SMOVL C00286 BC00286 V=100.0  +MOVJ EC00286
SREFP 3 C00287 BC00287  +REFP EC00287
CALL JOB:SEARCH-R1-S13D
SET P051 P006
SFTON3D P051
SMOVL C00288 BC00288 V=100.0  +MOVJ EC00288
SREFP 3 C00289 BC00289  +REFP EC00289
CALL JOB:SEARCH-R1-S13D
SET P051 P006
SFTON3D P051
SMOVL C00290 BC00290 V=100.0  +MOVJ EC00290
SMOVL C00291 BC00291 V=400.0  +MOVJ EC00291
MOVL C00292 BC00292 V=166.7  +MOVJ EC00292 VJ=100.00
MOVJ C00293 BC00293 VJ=100.00  +MOVJ EC00293 VJ=100.00
MOVJ C00294 BC00294 VJ=100.00  +MOVJ EC00294 VJ=100.00
MOVJ C00295 BC00295 VJ=100.00  +MOVJ EC00295 VJ=100.00
MOVJ C00296 BC00296 VJ=100.00  +MOVJ EC00296 VJ=100.00
MOVJ C00297 BC00297 VJ=100.00  +MOVJ EC00297 VJ=20.00
'Path S1445
SFTOF3D
MOVJ C00298 BC00298 VJ=100.00  +MOVJ EC00298 VJ=100.00
MOVL C00299 BC00299 V=666.7  +MOVJ EC00299 VJ=100.00
SMOVL C00300 BC00300 V=166.7  +MOVJ EC00300
SREFP 3 C00301 BC00301  +REFP EC00301
CALL JOB:SEARCH-R1-S13D
SET P070 P006
SFTON3D P070
SMOVL C00302 BC00302 V=166.7  +MOVJ EC00302
SMOVL C00303 BC00303 V=166.7  +MOVJ EC00303
SREFP 3 C00304 BC00304  +REFP EC00304
CALL JOB:SEARCH-R1-S13D
SET P070 P006
SFTON3D P070
SMOVL C00305 BC00305 V=166.7  +MOVJ EC00305
SFTOF3D
SMOVL C00306 BC00306 V=666.7  +MOVJ EC00306
SMOVL C00307 BC00307 V=166.7  +MOVJ EC00307
SREFP 3 C00308 BC00308  +REFP EC00308
CALL JOB:SEARCH-R1-S13D
SET P071 P006
SFTON3D P071
SMOVL C00309 BC00309 V=166.7  +MOVJ EC00309
SREFP 3 C00310 BC00310  +REFP EC00310
CALL JOB:SEARCH-R1-S13D
SET P071 P006
SFTON3D P071
SMOVL C00311 BC00311 V=166.7  +MOVJ EC00311
SMOVL C00312 BC00312 V=166.7  +MOVJ EC00312
SREFP 3 C00313 BC00313  +REFP EC00313
CALL JOB:SEARCH-R1-S13D
SET P071 P006
SFTON3D P071
SMOVL C00314 BC00314 V=166.7  +MOVJ EC00314
SFTOF3D
SMOVL C00315 BC00315 V=500.0  +MOVJ EC00315
SMOVL C00316 BC00316 V=166.7  +MOVJ EC00316
SREFP 3 C00317 BC00317  +REFP EC00317
CALL JOB:SEARCH-R1-S13D
SET P035 P006
SFTON3D P035
SMOVL C00318 BC00318 V=166.7  +MOVJ EC00318
SMOVL C00319 BC00319 V=166.7  +MOVJ EC00319
SREFP 3 C00320 BC00320  +REFP EC00320
CALL JOB:SEARCH-R1-S13D
SET P035 P006
SFTON3D P035
SMOVL C00321 BC00321 V=166.7  +MOVJ EC00321
SMOVL C00322 BC00322 V=166.7  +MOVJ EC00322
SMOVL C00323 BC00323 V=166.7  +MOVJ EC00323
SREFP 3 C00324 BC00324  +REFP EC00324
CALL JOB:SEARCH-R1-S13D
SET P035 P006
SFTON3D P035
SMOVL C00325 BC00325 V=166.7  +MOVJ EC00325
MOVL C00326 BC00326 V=666.7  +MOVJ EC00326 VJ=100.00
'Path S1446
SFTOF3D
MOVJ C00327 BC00327 VJ=100.00  +MOVJ EC00327 VJ=20.00
MOVJ C00328 BC00328 VJ=100.00  +MOVJ EC00328 VJ=100.00
MOVL C00329 BC00329 V=666.7  +MOVJ EC00329 VJ=100.00
SMOVL C00330 BC00330 V=166.7  +MOVJ EC00330
SREFP 3 C00331 BC00331  +REFP EC00331
CALL JOB:SEARCH-R1-S13D
SET P036 P006
SFTON3D P036
SMOVL C00332 BC00332 V=166.7  +MOVJ EC00332
SMOVL C00333 BC00333 V=166.7  +MOVJ EC00333
SMOVL C00334 BC00334 V=166.7  +MOVJ EC00334
SREFP 3 C00335 BC00335  +REFP EC00335
CALL JOB:SEARCH-R1-S13D
SET P036 P006
SFTON3D P036
SMOVL C00336 BC00336 V=166.7  +MOVJ EC00336
SMOVL C00337 BC00337 V=666.7  +MOVJ EC00337
SMOVL C00338 BC00338 V=666.7  +MOVJ EC00338
SMOVL C00339 BC00339 V=166.7  +MOVJ EC00339
SREFP 3 C00340 BC00340  +REFP EC00340
CALL JOB:SEARCH-R1-S13D
SET P036 P006
SFTON3D P036
SMOVL C00341 BC00341 V=166.7  +MOVJ EC00341
SMOVL C00342 BC00342 V=500.0  +MOVJ EC00342
'Path S1447
SFTOF3D
MOVJ C00343 BC00343 VJ=100.00  +MOVJ EC00343 VJ=20.00
MOVJ C00344 BC00344 VJ=100.00  +MOVJ EC00344 VJ=100.00
MOVL C00345 BC00345 V=500.0  +MOVJ EC00345 VJ=100.00
SMOVL C00346 BC00346 V=166.7  +MOVJ EC00346
SREFP 3 C00347 BC00347  +REFP EC00347
CALL JOB:SEARCH-R1-S13D
SET P033 P006
SFTON3D P033
SMOVL C00348 BC00348 V=166.7  +MOVJ EC00348
SREFP 3 C00349 BC00349  +REFP EC00349
CALL JOB:SEARCH-R1-S13D
SET P033 P006
SFTON3D P033
SMOVL C00350 BC00350 V=166.7  +MOVJ EC00350
MOVL C00351 BC00351 V=500.0  +MOVJ EC00351 VJ=100.00
MOVL C00352 BC00352 V=1000.0  +MOVJ EC00352 VJ=100.00
SMOVL C00353 BC00353 V=500.0  +MOVJ EC00353
'Path S1555
SFTOF3D
SMOVL C00354 BC00354 V=166.7  +MOVJ EC00354
SREFP 3 C00355 BC00355  +REFP EC00355
CALL JOB:SEARCH-R1-S13D
SET P053 P006
SFTON3D P053
SMOVL C00356 BC00356 V=166.7  +MOVJ EC00356
SREFP 3 C00357 BC00357  +REFP EC00357
CALL JOB:SEARCH-R1-S13D
SET P053 P006
SFTON3D P053
SMOVL C00358 BC00358 V=166.7  +MOVJ EC00358
SFTOF3D
SMOVL C00359 BC00359 V=1000.0  +MOVJ EC00359
SMOVL C00360 BC00360 V=166.7  +MOVJ EC00360
SREFP 3 C00361 BC00361  +REFP EC00361
CALL JOB:SEARCH-R1-S13D
SET P052 P006
SFTON3D P052
SMOVL C00362 BC00362 V=166.7  +MOVJ EC00362
SREFP 3 C00363 BC00363  +REFP EC00363
CALL JOB:SEARCH-R1-S13D
SET P052 P006
SFTON3D P052
SMOVL C00364 BC00364 V=166.7  +MOVJ EC00364
SFTOF3D
MOVJ C00365 BC00365 VJ=100.00  +MOVJ EC00365 VJ=100.00
MOVL C00366 BC00366 V=1000.0  +MOVJ EC00366 VJ=100.00
SMOVL C00367 BC00367 V=166.7  +MOVJ EC00367
SREFP 3 C00368 BC00368  +REFP EC00368
CALL JOB:SEARCH-R1-S13D
SET P032 P006
SFTON3D P032
SMOVL C00369 BC00369 V=166.7  +MOVJ EC00369
SMOVL C00370 BC00370 V=166.7  +MOVJ EC00370
SREFP 3 C00371 BC00371  +REFP EC00371
CALL JOB:SEARCH-R1-S13D
SET P032 P006
SFTON3D P032
SFTOF3D
SMOVL C00372 BC00372 V=166.7  +MOVJ EC00372
MOVL C00373 BC00373 V=666.7  +MOVJ EC00373 VJ=100.00
SMOVL C00374 BC00374 V=666.7  +MOVJ EC00374
SFTOF3D
SMOVL C00375 BC00375 V=166.7  +MOVJ EC00375
SREFP 3 C00376 BC00376  +REFP EC00376
CALL JOB:SEARCH-R1-S13D
SET P054 P006
SFTON3D P054
SMOVL C00377 BC00377 V=166.7  +MOVJ EC00377
SREFP 3 C00378 BC00378  +REFP EC00378
CALL JOB:SEARCH-R1-S13D
SET P054 P006
SFTON3D P054
SMOVL C00379 BC00379 V=166.7  +MOVJ EC00379
MOVL C00380 BC00380 V=1000.0  +MOVJ EC00380 VJ=100.00
'-90,0
'Path W1480
SFTOF3D
SFTON3D P032
MOVJ C00381 BC00381 VJ=100.00  +MOVJ EC00381 VJ=100.00
SMOVL C00382 BC00382 V=400.0  +MOVJ EC00382
SMOVL C00383 BC00383 V=166.7 PL=0  +MOVJ EC00383
SREFP 1 C00384 BC00384  +REFP EC00384
SREFP 2 C00385 BC00385  +REFP EC00385
MACRO1 MJ#(0) ARGF6
ARCON
SFTON3D P054
SMOVL C00386 BC00386 V=8.3  +MOVJ EC00386
SMOVL C00387 BC00387 V=8.3  +MOVJ EC00387
ARCOF
SFTOF3D
SMOVL C00388 BC00388 V=400.0  +MOVJ EC00388
SMOVL C00389 BC00389 V=1000.0  +MOVJ EC00389
'Path W1481
SFTOF3D
SFTON3D P035
MOVJ C00390 BC00390 VJ=100.00  +MOVJ EC00390 VJ=100.00
SMOVL C00391 BC00391 V=400.0  +MOVJ EC00391
SMOVL C00392 BC00392 V=133.3 PL=0  +MOVJ EC00392
SREFP 1 C00393 BC00393  +REFP EC00393
SREFP 2 C00394 BC00394  +REFP EC00394
MACRO1 MJ#(0) ARGF14
ARCON
SMOVL C00395 BC00395 V=8.3  +MOVJ EC00395
SFTON3D P052
SMOVL C00396 BC00396 V=8.3  +MOVJ EC00396
SMOVL C00397 BC00397 V=8.3  +MOVJ EC00397
ARCOF
SFTOF3D
SMOVL C00398 BC00398 V=400.0  +MOVJ EC00398
SMOVL C00399 BC00399 V=1000.0  +MOVJ EC00399
SFTOF3D
MOVJ C00400 BC00400 VJ=100.00  +MOVJ EC00400 VJ=100.00
'Path W1482
SFTOF3D
MOVJ C00401 BC00401 VJ=100.00  +MOVJ EC00401 VJ=100.00
SMOVL C00402 BC00402 V=400.0  +MOVJ EC00402
SFTON3D P070
SMOVL C00403 BC00403 V=133.3 PL=0  +MOVJ EC00403
SREFP 1 C00404 BC00404  +REFP EC00404
SREFP 2 C00405 BC00405  +REFP EC00405
MACRO1 MJ#(0) ARGF9
ARCON
SMOVL C00406 BC00406 V=10.8  +MOVJ EC00406
SFTON3D P071
SMOVL C00407 BC00407 V=10.3  +MOVJ EC00407
SMOVL C00408 BC00408 V=10.3  +MOVJ EC00408
ARCOF
SMOVL C00409 BC00409 V=400.0  +MOVJ EC00409
SMOVL C00410 BC00410 V=1000.0  +MOVJ EC00410
SFTOF3D
'Path W1483
SFTOF3D
SFTON3D P021
MOVJ C00411 BC00411 VJ=100.00  +MOVJ EC00411 VJ=100.00
SMOVL C00412 BC00412 V=166.7 PL=0  +MOVJ EC00412
SREFP 1 C00413 BC00413  +REFP EC00413
SREFP 2 C00414 BC00414  +REFP EC00414
MACRO1 MJ#(0) ARGF14
ARCON
SMOVL C00415 BC00415 V=8.3  +MOVJ EC00415
SMOVL C00416 BC00416 V=8.3  +MOVJ EC00416
SMOVL C00417 BC00417 V=8.3  +MOVJ EC00417
ARCOF
SMOVL C00418 BC00418 V=400.0  +MOVJ EC00418
SMOVL C00419 BC00419 V=1000.0  +MOVJ EC00419
SFTOF3D
'Path W1484
SFTOF3D
SFTON3D P036
MOVJ C00420 BC00420 VJ=100.00  +MOVJ EC00420 VJ=100.00
SMOVL C00421 BC00421 V=400.0  +MOVJ EC00421
SMOVL C00422 BC00422 V=133.3 PL=0  +MOVJ EC00422
SREFP 1 C00423 BC00423  +REFP EC00423
SREFP 2 C00424 BC00424  +REFP EC00424
MACRO1 MJ#(0) ARGF6
ARCON
SMOVL C00425 BC00425 V=12.5  +MOVJ EC00425
ARCOF
SFTOF3D
SMOVL C00426 BC00426 V=400.0  +MOVJ EC00426
SMOVL C00427 BC00427 V=1000.0  +MOVJ EC00427
SFTOF3D
'Path W1485
SFTOF3D
SFTON3D P033
MOVJ C00428 BC00428 VJ=100.00  +MOVJ EC00428 VJ=100.00
SMOVL C00429 BC00429 V=400.0  +MOVJ EC00429
SMOVL C00430 BC00430 V=133.3 PL=0  +MOVJ EC00430
SREFP 1 C00431 BC00431  +REFP EC00431
SREFP 2 C00432 BC00432  +REFP EC00432
MACRO1 MJ#(0) ARGF14
ARCON
SMOVL C00433 BC00433 V=10.0  +MOVJ EC00433
SMOVL C00434 BC00434 V=10.0  +MOVJ EC00434
ARCOF
SMOVL C00435 BC00435 V=10.8  +MOVJ EC00435
ARCON
SMOVL C00436 BC00436 V=10.0  +MOVJ EC00436
SFTON3D P053
SMOVL C00437 BC00437 V=10.0  +MOVJ EC00437
SMOVL C00438 BC00438 V=10.0  +MOVJ EC00438
ARCOF
SFTOF3D
SMOVL C00439 BC00439 V=400.0  +MOVJ EC00439
SMOVL C00440 BC00440 V=1000.0  +MOVJ EC00440
SFTOF3D
'Path W1486
SFTOF3D
SFTON3D P036
MOVJ C00441 BC00441 VJ=100.00  +MOVJ EC00441 VJ=20.00
MOVJ C00442 BC00442 VJ=100.00  +MOVJ EC00442 VJ=100.00
SMOVL C00443 BC00443 V=500.0  +MOVJ EC00443
SMOVL C00444 BC00444 V=166.7 PL=0  +MOVJ EC00444
SREFP 1 C00445 BC00445  +REFP EC00445
SREFP 2 C00446 BC00446  +REFP EC00446
MACRO1 MJ#(0) ARGF6
ARCON
SMOVL C00447 BC00447 V=10.8  +MOVJ EC00447
SMOVL C00448 BC00448 V=10.8  +MOVJ EC00448
ARCOF
SMOVL C00449 BC00449 V=400.0  +MOVJ EC00449
SMOVL C00450 BC00450 V=1000.0  +MOVJ EC00450
SFTOF3D
MOVJ C00451 BC00451 VJ=100.00  +MOVJ EC00451 VJ=100.00
MOVJ C00452 BC00452 VJ=100.00  +MOVJ EC00452 VJ=100.00
MOVJ C00453 BC00453 VJ=100.00  +MOVJ EC00453 VJ=100.00
MOVJ C00454 BC00454 VJ=100.00  +MOVJ EC00454 VJ=100.00
MOVJ C00455 BC00455 VJ=100.00  +MOVJ EC00455 VJ=100.00
'Path W1465
SFTOF3D
SFTON3D P037
SMOVL C00456 BC00456 V=400.0  +MOVJ EC00456
SMOVL C00457 BC00457 V=133.3 PL=0  +MOVJ EC00457
SREFP 1 C00458 BC00458  +REFP EC00458
SREFP 2 C00459 BC00459  +REFP EC00459
MACRO1 MJ#(0) ARGF14
ARCON
SFTON3D P050
SMOVL C00460 BC00460 V=8.3  +MOVJ EC00460
SMOVL C00461 BC00461 V=8.3  +MOVJ EC00461
ARCOF
SMOVL C00462 BC00462 V=250.0  +MOVJ EC00462
SFTOF3D
MOVJ C00463 BC00463 VJ=100.00  +MOVJ EC00463 VJ=100.00
MOVJ C00464 BC00464 VJ=100.00  +MOVJ EC00464 VJ=100.00
MOVJ C00465 BC00465 VJ=100.00  +MOVJ EC00465 VJ=100.00
MOVJ C00466 BC00466 VJ=100.00  +MOVJ EC00466 VJ=100.00
MOVJ C00467 BC00467 VJ=100.00  +MOVJ EC00467 VJ=100.00
'Path W1469
SFTOF3D
SFTON3D P039
SMOVL C00468 BC00468 V=400.0  +MOVJ EC00468
SMOVL C00469 BC00469 V=133.3 PL=0  +MOVJ EC00469
SREFP 1 C00470 BC00470  +REFP EC00470
SREFP 2 C00471 BC00471  +REFP EC00471
MACRO1 MJ#(0) ARGF14
ARCON
SFTON3D P051
SMOVL C00472 BC00472 V=8.3  +MOVJ EC00472
SMOVL C00473 BC00473 V=8.3  +MOVJ EC00473
ARCOF
SMOVL C00474 BC00474 V=83.3  +MOVJ EC00474
SMOVL C00475 BC00475 V=133.3  +MOVJ EC00475
SFTOF3D
MOVJ C00476 BC00476 VJ=100.00  +MOVJ EC00476 VJ=100.00
MOVJ C00477 BC00477 VJ=100.00  +MOVJ EC00477 VJ=100.00
MOVJ C00478 BC00478 VJ=100.00  +MOVJ EC00478 VJ=100.00
MOVJ C00479 BC00479 VJ=100.00  +MOVJ EC00479 VJ=100.00
MOVJ C00480 BC00480 VJ=100.00  +MOVJ EC00480 VJ=20.00
END
